(* PLC project Base_Elements, Beckhoff Automation GmbH TwinCAT PLC Control 3.5.6.0 *)
(* stored: creationDateTime 2015-09-07T10:33:48.4706416, modificationDateTime 2015-09-07T10:33:48.472642 *)

TYPE E_ADS_AccessType : (READ := 0, WRITE := 1);
END_TYPE

TYPE T_ADS_ConnectionData : STRUCT
  udiConID : UDINT;  (* Connection ID. Automatically assigned by calling method for adding new connection *)
  udiHandle : UDINT;  (* Handle ID for data exchange. Determined automatically during state PONbusy. *)
  strRoute : STRING;  (* Route of the PRG or FUB instance on server side. Example: 'SlowPRG_1.fbData.SIf.cur.st_ADSData' *)
  uinTargetPort : UINT;  (* ADS target port *)
  strNetID : STRING(30);  (* NetID *)
  eAccessType : E_ADS_AccessType;  (* Access type *)
  udiDataLen : UDINT;  (* Length of the data structure *)
  pData : PVOID;  (* Pointer to data structure. Note: Defined structure must be the same on client and server side. *)
END_STRUCT;
END_TYPE

TYPE T_Ctrl_SIf_ACL : STRUCT
  Par : T_Ctrl_SIf_ACL_Par;  (* parameter *)
  Cur : T_Ctrl_SIf_ACL_Cur;  (* current values *)
  Alm : ARRAY[1..7] OF T_Ctrl_Alm;  (* alarm number used in this controller *)
END_STRUCT;
END_TYPE

TYPE T_Ctrl_SIf_ACL_Cur : STRUCT
  uinNumOfAdsConnections : UINT;  (* Shows the number of ADS (server) connections *)
END_STRUCT;
END_TYPE

TYPE T_Ctrl_SIf_ACL_Par : STRUCT
  udiTOPowerOn_ms : UDINT;  (* [ms] Timeout power on. Timeout for initialize all ADS connections. *)
  udiTOAddRoute_ms : UDINT;  (* [ms] Timeout add route *)
  udiTOReadData_ms : UDINT;  (* [ms] Timeout read data *)
  udiTOWriteData_ms : UDINT;  (* [ms] Timeout write data *)
  udiTORWData_ms : UDINT;  (* [ms] Timeout read/write data *)
  udiPollingInterval_ms : UDINT;  (* [ms] Polling interval for read/write of all ADS connections in list *)
END_STRUCT;
END_TYPE

TYPE E_BCD_Type : (None := 0, SICK, KEYENCE);
END_TYPE

TYPE T_BCD : STRUCT
  strState : STRING;
  strCmd : STRING;
  intCmd : INT;
  stStatus : T_BCD_Status;
  stErr : T_BCD_Error;
  stCfg : T_BCD_Cfg;
  stPar : T_BCD_Par;
  stData : T_BCD_Data;
END_STRUCT;
END_TYPE

TYPE T_BCD_Cfg : STRUCT
  bolSimulation : BOOL;
  strSensorIPAdr : STRING(15) := '';
  udiSensorPort : UDINT := 0;
  iSensorType : E_BCD_Type;
  bolResponseIncludingDiagnostics : BOOL;  (* Barcode is also sending diagnostics data *)
END_STRUCT;
END_TYPE

TYPE T_BCD_Data : STRUCT
  bolCodeReaded : BOOL;
  uliBarCode : ULINT;
  strBarCode : STRING;
  stDevInfo : T_BCD_DeviceInfo;
  stServInfo : T_BCD_ServiceInfo;
  stOpData : T_BCD_OperatingData;
END_STRUCT;
END_TYPE

TYPE T_BCD_DeviceInfo : STRUCT
  strComTestResult : STRING(40);
  strManufacturer : STRING(25);
  strDeviceType : STRING(25);
  strOrderNumber : STRING(20);
  strSWVersion : STRING(10);
  strFWVersion : STRING(10);  (* shows the firmware version of the device *)
  strSerialNumber : STRING(20);
END_STRUCT;
END_TYPE

TYPE T_BCD_Error : STRUCT
  bolErrAck : BOOL;  (* Reset failure *)
  bolErrorActive : BOOL;  (* atleast one failure active *)
  bolSocketError : BOOL;  (* error in TCP socket *)
  bolSensorError : BOOL;  (* error in sensor (SICK) *)
  udiErrorID : UDINT;  (* error ID *)
END_STRUCT;
END_TYPE

TYPE T_BCD_OperatingData : STRUCT
  strPowerOnCounter : STRING(25);
  strOpHours : STRING(25);
  strPowerOnHours : STRING(20);
END_STRUCT;
END_TYPE

TYPE T_BCD_Par : STRUCT
  tTOConnection : TIME;
  tTOSend : TIME;
  tTOReceive : TIME;
END_STRUCT;
END_TYPE

TYPE T_BCD_ServiceInfo : STRUCT
  strLastUsername : STRING(25);
  strLastParChangeDate : STRING(10);
  strLastParChangeTime : STRING(5);
END_STRUCT;
END_TYPE

TYPE T_BCD_StateMachine : STRUCT
  intState : INT;  (* actual state *)
  intStateLastCycle : INT;  (* state of last cycle *)
  intStateHistory : INT;  (* save history backup p.e. in ERROR state *)
  intStateNext : INT;  (* set state for next cycle *)
  udiTimeInState_ms : UDINT;  (* Time in this State *)
END_STRUCT;
END_TYPE

TYPE T_BCD_Status : STRUCT
  bolSocketConnected : BOOL;  (* Socket connected *)
  bolComChecked : BOOL;
END_STRUCT;
END_TYPE

TYPE T_BCD_TxStructure : STRUCT
  intMessageSize : UINT;  (* Actual message size *)
  aTxData : ARRAY[0..300] OF BYTE;  (* Tx data buffer *)
END_STRUCT;
END_TYPE

TYPE E_ALM_PRS : (Dummy := 1, MAX_E_ALM_PRS) UINT;
END_TYPE

TYPE T_Ctrl_SIf_PRS : STRUCT
  Cfg : T_Ctrl_SIf_PRS_Cfg;  (* configuration *)
  Par : T_Ctrl_SIf_PRS_Par;  (* parameter *)
  Cur : T_Ctrl_SIf_PRS_Cur;  (* current values *)
  In : T_Ctrl_SIf_PRS_In;  (* io input *)
  Out : T_Ctrl_SIf_PRS_Out;  (* io output *)
  Alm : ARRAY[1..E_ALM_PRS.MAX_E_ALM_PRS] OF T_Ctrl_Alm;  (* alarm number used in this controller *)
  Ilk : T_Ctrl_SIf_PRS_Ilk;  (* interlock of output/movements *)
END_STRUCT;
END_TYPE

TYPE T_Ctrl_SIf_PRS_Cfg : STRUCT

END_STRUCT;
END_TYPE

TYPE T_Ctrl_SIf_PRS_Cur : STRUCT

END_STRUCT;
END_TYPE

TYPE T_Ctrl_SIf_PRS_Ilk : STRUCT

END_STRUCT;
END_TYPE

TYPE T_Ctrl_SIf_PRS_In : STRUCT
  bolPresent : BASE_PLC.T_Ctrl_IoBool;  (* Input Sensor is present *)
END_STRUCT;
END_TYPE

TYPE T_Ctrl_SIf_PRS_Out : STRUCT

END_STRUCT;
END_TYPE

TYPE T_Ctrl_SIf_PRS_Par : STRUCT
  udiDebouncePresentTime_ms : UDINT;  (* [ms] Debounce time until it shows as present *)
  udiDebounceAbsentTime_ms : UDINT;  (* [ms] Debounce time until it shows as absent *)
  bolSimHangerAvailable : BOOL;  (* True = simulated hanger available *)
END_STRUCT;
END_TYPE

TYPE E_Typ_Baudrate : (baud_2400 := 4, baud_4800 := 5, baud_9600 := 6, baud_19200 := 7, baud_38400 := 8, baud_57600 := 9, baud_115200 := 10);
END_TYPE

(* values of E_Typ_Ftim: RF300: Setting for air interface *)

TYPE E_Typ_Ftim : (RF300 := 0, ISO_generall := 1, ISO_infineon := 3, ISO_Fujitsu := 4, ISO_NXP := 5, ISO_TI := 6, ISO_ST := 7, Max_E_Typ_Ftim);
END_TYPE

TYPE T_RFD : STRUCT
  strState : STRING;
  strCmd : STRING;
  intCmd : INT;
  intServiceCmd : INT;
  stStatus : T_RFD_Status;
  stCfg : T_RFD_Cfg;
  stCur : T_RFD_Cur;
  stErr : T_RFD_Error;
END_STRUCT;
END_TYPE

TYPE T_RFD_Cfg : STRUCT
  bolSimulation : BOOL;
  eTyp : E_Typ_RFW;
  usiResetParameter : USINT := 2#101010;  (* Reset parameter value *)
  usiFtimSetting : E_Typ_Ftim;  (* Setting of the Air interface *)
  usiResetOption1 : USINT := 2#10;  (* Reset option1 value *)
  uinBaudrate : USINT;  (* Set Baudrate *)
  uinComSettings : USINT;  (* Set Communikationsettings *)
  stNetId : TC2_SYSTEM.T_AmsNetID;  (* Net ID oft EtherCat Master *)
  uinSlaveAddr : UINT;  (* Port Number of EtherCat Slave Comunication Module *)
  uinCoeIndexComSettings : WORD := 16#8000;  (* CoE Object Index for Communication Settings *)
  usiCoeSubindexComBaudrate : BYTE := 16#11;  (* CoE Object SubIndex for Baudrate *)
  usiCoeSubindexComDataframe : BYTE := 16#15;  (* CoE Object SubIndex for Dataframe *)
  udiRetry : UDINT := 10;  (* Retry Job to RFID Reader *)
  usiMemory : USINT := 0;  (* /////////////////////////////////////////////// Reset Memory 00=RAM, 01=remanent *)
  usiScanMode : USINT := 1;  (* Scan Mode 00= Continous Read; 01=Single Read *)
  uinLockTime_ms : UINT := 5000;  (* Lock Time in ms *)
END_STRUCT;
END_TYPE

TYPE T_RFD_Cur : STRUCT
  pData : POINTER TO ARRAY[0..255] OF BYTE;  (* Pointer to Received Data Array *)
  uinAdressData : UINT;  (* Startadress to Read/Write at the data Array Element *)
  uinAdressTag : UINT;  (* Startadress to Read/Write at the Tag *)
  usiCount : USINT;  (* Number of bytes to Read/Write *)
END_STRUCT;
END_TYPE

TYPE T_RFD_Error : STRUCT
  bolErrAck : BOOL;  (* Reset failure *)
  bolErrorActive : BOOL;  (* atleast one failure active *)
  bolComError : BOOL;  (* error at communication card *)
  bolProtcolError : BOOL;
  bolRFIDError : BOOL;  (* Error with RF ID Tag *)
  bolSDOError : BOOL;  (* Error at setting of the communication Card (SDO Write) *)
  udiErrorID : UDINT;  (* information to Communication Card error *)
END_STRUCT;
END_TYPE

TYPE T_RFD_MDS_Diagnose : STRUCT
  usiLFD : USINT;  (* Power flux density: as smaller the value, as higher the field intensity *)
  usiFZP : USINT;  (* Errorcounter inactive mode *)
  usiFZA : USINT;  (* Errorcounter active: CRC or signature errors *)
  usiANWZ : USINT;  (* Presence time of tag, resolution in 9.7ms *)
END_STRUCT;
END_TYPE

TYPE T_RFD_MDS_State : STRUCT
  bytMDSType : BYTE;  (* MDS Type 1=no FRAM; 2=8k FRAM; 3=32k FRAM; 4=64k FRAM; 5=128k FRAM; 6=256k FRAM *)
  bytLockState : BYTE;  (* Lock bit registers (lock state) *)
  bytVersion : BYTE;  (* MDS Version *)
  worMemSize : WORD;  (* Memory Size *)
  bytBlockSize : BYTE;  (* Blocksize in Byte *)
  bytBlockNo : BYTE;  (* Value of memory Blocks *)
END_STRUCT;
END_TYPE

TYPE T_RFD_SLG_Diagnose : STRUCT
  usiS_Info : USINT;  (* Mode SLG Diagnose *)
  usiFZP : USINT;  (* Errorcounter inactive mode *)
  usiABZ : USINT;  (* Counter abort *)
  usiCFZ : USINT;  (* Errorcounter code errors *)
  usiSFZ : USINT;  (* Errorcounter signature errors *)
  usiCRCFZ : USINT;  (* Errorcounter CRC *)
  usiBSTAT : USINT;  (* Actual command state *)
  usiASMFZ : USINT;  (* Counter interface errors to host (Parity, BCC, Frame) *)
END_STRUCT;
END_TYPE

TYPE T_RFD_SLG_State : STRUCT
  bytHWType : BYTE;  (* HW Type of SLG 0=RF310R RF340R RF350R (-xAA10); 1=RF380R (-3AA10); 2=RF310R(-1AB10); 3=RF380R (-3AB10); 4=RF340R RF350R (-2AB10,-4AB10) *)
  worHWVersion : WORD;  (* HW Version *)
  worURLVersion : WORD;  (* Loading Version *)
  bytFWType : BYTE;  (* FW Type *)
  worFWVersion : WORD;  (* FW Version *)
  bytDriverType : BYTE;  (* Driver Type 1=3964R *)
  worDriverVersion : WORD;  (* Driver Version *)
  bytComm : BYTE;  (* Communication port 1=RS422, 2=RS232 *)
  bytBaud : BYTE;  (* Communication Baud rate 1=19.2kBaud; 3=57.6kBaud; 5=115.2kBaud *)
  bytPower : BYTE;  (* sending power (only RF380R) 0=standard; 2=0.5W; 3=0.75W; 4=1W; 5=1.25W (default); 6=1.5W; 7=1.75W; 8=2W *)
  bytMtag : BYTE;  (* Number of maximal tags in the field *)
  bytFtim : BYTE;  (* air interface 0=RF300; 1=ISO generall; 3=ISO infineon Chip; 4=ISO Fujitsu; 5=ISO NXP; 6=ISO TI; 7=ISO ST *)
  bytAntenna : BYTE;  (* State antenna 1=ON; 2=OFF *)
  bytPresence : BYTE;  (* Tag presence 0=No presence; 1=prexence *)
END_STRUCT;
END_TYPE

TYPE T_RFD_StateMachine : STRUCT
  intState : INT;  (* actual state *)
  intStateLastCycle : INT;  (* state of last cycle *)
  intStateHistory : INT;  (* save history backup p.e. in ERROR state *)
  intStateNext : INT;  (* set state for next cycle *)
  udiTimeInState_ms : UDINT;  (* Time in this State *)
END_STRUCT;
END_TYPE

TYPE T_RFD_Status : STRUCT
  bolStartupOk : BOOL;  (* 1 = Antenna is initialized *)
  bolInitOk : BOOL;  (* 1 = Antenna is initialized *)
  bolOn : BOOL;  (* 1 = Antenna is on *)
  bolPresent : BOOL;  (* 1 = tag is present *)
  bolL_UEB : BOOL;  (* 1 = Communication to SLG is OK *)
  stSLG_State : T_RFD_SLG_State;  (* SLG State only actual on demand *)
  stSLG_Diag : T_RFD_SLG_Diagnose;  (* SLG Diagnose only actual on demand *)
  stMDS_State : T_RFD_MDS_State;  (* SLG State only actual on demand *)
  stMDS_Diag : T_RFD_MDS_Diagnose;  (* SLG Diagnose only actual on demand *)
  abyteUID : ARRAY[0..7] OF BYTE;  (* Tag ID *)
END_STRUCT;
END_TYPE

TYPE T_StateWord : STRUCT
  bolTransmitAccepted : BOOL;  (* Acknowledge the datachange of this Command bit *)
  bolReceiveRequest : BOOL;  (* New Datat at the input *)
  bolInputAccepted : BOOL;  (* 0=Ready for Data exchange; 1=initialisation of the clam *)
  bolBufferFull : BOOL;  (* Input Buffer is full, all new arriveing data lost *)
  bolParityErr : BOOL;  (* Parity Error occured *)
  bolFramingErr : BOOL;  (* Framing Error occured *)
  bolOverrunErr : BOOL;  (* Overrun Error occured *)
  usiInLenght : USINT;  (* Amounth of the reached Input Bytes *)
END_STRUCT;
END_TYPE

TYPE E_LIGHTSTATE : (Off, BlinkSlow, BlinkFast, On);
END_TYPE

TYPE E_StackLightColor : (Red, Yellow, Green, Blue, Max_SackLightColor);
END_TYPE

TYPE T_LighInformation : STRUCT
  eState : E_LIGHTSTATE;
  udiTime_ms : UDINT;
  bolOutput : REFERENCE TO REFERENCE TO BOOL;
END_STRUCT;
END_TYPE

TYPE T_BCC_Data : STRUCT
  uliBarCode : ULINT;
  strBarCode : STRING;
END_STRUCT;
END_TYPE

TYPE T_Ctrl_SIf_BCC : STRUCT
  Cfg : T_Ctrl_SIf_BCC_Cfg;  (* configuration *)
  Par : T_Ctrl_SIf_BCC_Par;  (* parameter *)
  Cur : T_Ctrl_SIf_BCC_Cur;  (* current values *)
  In : T_Ctrl_SIf_BCC_In;  (* io input *)
  Out : T_Ctrl_SIf_BCC_Out;  (* io output *)
  Alm : ARRAY[1..7] OF T_Ctrl_Alm;  (* alarm number used in this controller *)
END_STRUCT;
END_TYPE

TYPE T_Ctrl_SIf_BCC_Cfg : STRUCT
  strSensorIPAdr : STRING(15) := '';  (* IP Adress of the sensor (PLC = Client, Sensor = Server) *)
  udiSensorPort : UDINT := 0;  (* Port number of the sensor *)
  iSensorType : E_BCD_Type;
END_STRUCT;
END_TYPE

TYPE T_Ctrl_SIf_BCC_Cur : STRUCT
  bolConnected : BOOL;  (* Sensor connected *)
  bolComChecked : BOOL;  (* Communication checked during PON *)
  bolNewCodeReaded : BOOL;  (* 1 = new bar code readed *)
  bolNoRead : BOOL;  (* 1 = no code readed, answer *No Read* *)
  stData : T_BCC_Data;  (* Sensor data *)
END_STRUCT;
END_TYPE

TYPE T_Ctrl_SIf_BCC_In : STRUCT
  bolSensorTrigScan : BASE_PLC.T_Ctrl_IoBool;  (* Sensor input for triggering a new barcode scan *)
END_STRUCT;
END_TYPE

TYPE T_Ctrl_SIf_BCC_Out : STRUCT

END_STRUCT;
END_TYPE

TYPE T_Ctrl_SIf_BCC_Par : STRUCT
  udiTOPowerOn_ms : UDINT;  (* [ms] Timeout power on *)
  udiTORead_ms : UDINT;  (* [ms] Timeout read *)
  udiExecuteScanDelayTime_ms : UDINT;  (* [ms] Barcode scan delay time - Delay before a barcode scan will be triggered after a new product has been detected by trigger sensor input *)
END_STRUCT;
END_TYPE

{attribute 'qualified_only'}
TYPE E_ALM_CYL : (SensorRetractAlwaysOn := 1, SensorExtendNotReached := 2, SensorExtendAlwaysOn := 3, SensorRetractNotReached := 4, InterlockExtend := 5, InterlockRetract := 6, MAX_E_ALM) UINT;
END_TYPE

(* values of E_Typ_CYL: Valve2_Sensor2: bistabile and two feedback sensors; Valve2_SensorExtended: bistabile and extended feedback sensors; Valve2_SensorRetracted: bistabile and retracted feedback sensors; Valve2_Sensor0: bistabile and no feedback sensors; Valve1_Sensor2: monostabile and 2 feedback sensors; Valve1_SensorExtended: monostabile and extended feedback sensors; Valve1_SensorRetracted: monostabile and retracted feedback sensor; Valve1_Sensor0: monostabile and no feedback sensors *)

TYPE E_Typ_CYL : (Valve2_Sensor2 := 0, Valve2_SensorExtended, Valve2_SensorRetracted, Valve2_Sensor0, Valve1_Sensor2, Valve1_SensorExtended, Valve1_SensorRetracted, Valve1_Sensor0, Max_E_Typ_CYL);
END_TYPE

TYPE T_Ctrl_SIf_CYL : STRUCT
  Cfg : T_Ctrl_SIf_CYL_Cfg;  (* configuration *)
  Par : T_Ctrl_SIf_CYL_Par;  (* parameter *)
  Cur : T_Ctrl_SIf_CYL_Cur;  (* current values *)
  In : T_Ctrl_SIf_CYL_In;  (* io input *)
  Out : T_Ctrl_SIf_CYL_Out;  (* io output *)
  Alm : ARRAY[1..(E_ALM_CYL.MAX_E_ALM - 1)] OF T_Ctrl_Alm;  (* alarm number used in this controller *)
  Ilk : T_Ctrl_SIf_CYL_Ilk;  (* interlock of output/movements *)
END_STRUCT;
END_TYPE

TYPE T_Ctrl_SIf_CYL_Cfg : STRUCT
  eTyp : E_Typ_CYL;
END_STRUCT;
END_TYPE

TYPE T_Ctrl_SIf_CYL_Cur : STRUCT
  udiMoveTimeRetract : UDINT;  (* [ms] time last movement to retract *)
  udiMoveTimeExtend : UDINT;  (* [ms] time last movement to extend *)
END_STRUCT;
END_TYPE

TYPE T_Ctrl_SIf_CYL_Ilk : STRUCT
  bolRetract : BOOL;  (* interlock retraction of cylinder *)
  bolExtend : BOOL;  (* interlock extend of cylinder *)
END_STRUCT;
END_TYPE

TYPE T_Ctrl_SIf_CYL_In : STRUCT
  bolExtended : T_Ctrl_IoBool;  (* sensor feedback position extended reached *)
  bolRetracted : T_Ctrl_IoBool;  (* sensor feedback position retracted reached *)
END_STRUCT;
END_TYPE

TYPE T_Ctrl_SIf_CYL_Out : STRUCT
  bolRetract : T_Ctrl_IoBool;  (* switch valve retract *)
  bolExtend : T_Ctrl_IoBool;  (* switch valve extend *)
END_STRUCT;
END_TYPE

TYPE T_Ctrl_SIf_CYL_Par : STRUCT
  udiExtendTime_ms : UDINT;  (* [ms] until failure to long time for extend *)
  udiRetractTime_ms : UDINT;  (* [ms] until failure to long time for retract *)
  udiSimExtendTime_ms : UDINT;  (* [ms] simulation time for extend or /2 of timeout time? *)
  udiSimRetractTime_ms : UDINT;  (* [ms] simulation time for retract or /2 of timeout time? *)
END_STRUCT;
END_TYPE

TYPE E_Typ_DRV : (None := 0, TLP, TLK, TLKV, TLPsort, TLS, TLC, Max_E_Typ_JUN);
END_TYPE

TYPE T_Ctrl_SIf_DRV : STRUCT
  Cfg : T_Ctrl_SIf_DRV_Cfg;  (* configuration *)
  Par : T_Ctrl_SIf_DRV_Par;  (* parameter *)
  Cur : T_Ctrl_SIf_DRV_Cur;  (* current values *)
  In : T_Ctrl_SIf_DRV_In;  (* io input *)
  Out : T_Ctrl_SIf_DRV_Out;  (* io output *)
  Alm : ARRAY[1..5] OF T_Ctrl_Alm;  (* alarm number used in this controller *)
END_STRUCT;
END_TYPE

TYPE T_Ctrl_SIf_DRV_Cfg : STRUCT
  eTyp : E_Typ_DRV;  (* Type of drive *)
  dinDistPerPulse_um : DINT;  (* Distance per pulse *)
  bolSpeedVariable : BOOL;  (* Has Variable Speed *)
  bolPulseExist : BOOL;  (* Has Pulse signal for position and speed calculation *)
  usiCountBlockedSupervis : USINT;  (* Number of blocked supervision inputs *)
  dinPinDistance_um : DINT;  (* [um] PinDistance *)
  bolEnableMaintenaceSwitch : BOOL;  (* Enable Maintenace Switch *)
END_STRUCT;
END_TYPE

TYPE T_Ctrl_SIf_DRV_Cur : STRUCT
  dinPulseCounter : DINT;
  dinPos_um : DINT;
  dinSpeed_um_s : DINT;
END_STRUCT;
END_TYPE

TYPE T_Ctrl_SIf_DRV_In : STRUCT
  bolOverload : T_Ctrl_IoBool;
  bolPulse : T_Ctrl_IoBool;
  a_bolBlockedSupvervis : ARRAY[1..cMAX_BLOCKED_SUP] OF BASE_PLC.T_Ctrl_IoBool;
  bolMaintenanceSwitch : T_Ctrl_IoBool;  (* DI of Maintenance Switch *)
END_STRUCT;
END_TYPE

TYPE T_Ctrl_SIf_DRV_Out : STRUCT
  bolSpeed_1 : T_Ctrl_IoBool;  (* bolSpeed_1 = slow bolSpeed_2 = fast bolSpeed_1 & bolSpeed_2 = middle speed *)
  bolSpeed_2 : T_Ctrl_IoBool;
END_STRUCT;
END_TYPE

TYPE T_Ctrl_SIf_DRV_Par : STRUCT
  udi_pulseTimeout_ms : UDINT;  (* [ms] Timeout supervision of pulse in RUN *)
  udi_pulseSim_ms : UDINT;  (* [ms] Simulation of pulse in RUN: 0.676mm/ms / 38.4mm/puls => 56.8ms/puls *)
  usi_speedLevel : USINT;  (* 0=slow, 1=middle, 2=fast *)
  int_MaxBrokenPins : INT;  (* Maximum Broken Pins *)
END_STRUCT;
END_TYPE

(* values of E_ALM_ECD: ADS_ComError: ADS Communication Error to EtherCAT Master => Info = ADS_Errorcode; TimeOutFunction: A Function is not finished after the defined Timeout; NotAllSlaveConnected: Configured and reached Slaves are not the same => Info Byte 0+1 = Slave Addres from last error Info Byte 2+3 = Numbers of error Slaves; ToManySlaves: More slaves at the master as the structure could handle => Info Byte 0+1 = Slave Addres from last error Info Byte 2+3 = Numbers of error Slaves; MasterStateError: Master not in the correct state => Info = Masterstate; SlaveStateError: Minimum one Slave not in the correct state => Byte 0+1 = Slave Addres from last error, Info Byte 2 + 3 = State of last error Slave; SlaveCRCError: Minimum one Slave has to many CRC Erros => Byte 0+1 = Slave Addres from last error, Info Byte 2 +3 = Number of CRC Errors from last Slave with error; SlaveLinkError: Minimum one Slave has a LinkState Erros => Byte 0+1 = Slave Addres from last error Info Byte 2 + 3 = Link State of last error Slave; NoSlaveFound: No slave found in the network; StateChanges: To many abnormal State Changes *)

TYPE E_ALM_ECD : (ADS_ComError := 1, TimeOutFunction := 2, NotAllSlaveConnected := 3, ToManySlaves := 4, MasterStateError := 5, SlaveStateError := 6, SlaveCRCError := 7, SlaveLinkError := 8, NoSlaveFound := 9, StateChanges := 10, MAX_E_ALM) UINT;
END_TYPE

TYPE T_Ctrl_SIf_ECD : STRUCT
  Cfg : T_Ctrl_SIf_ECD_Cfg;  (* configuration *)
  Par : T_Ctrl_SIf_ECD_Par;  (* parameter *)
  Cur : T_Ctrl_SIf_ECD_Cur;  (* current values *)
  Alm : ARRAY[1..(E_ALM_ECD.MAX_E_ALM - 1)] OF T_Ctrl_Alm;  (* alarm number used in this controller *)
END_STRUCT;
END_TYPE

TYPE T_Ctrl_SIf_ECD_Cfg : STRUCT
  strNetID : STRING(30);  (* NetID *)
  bolRunAlways : BOOL;  (* Run allways the scanning without set into run *)
END_STRUCT;
END_TYPE

TYPE T_Ctrl_SIf_ECD_Cur : STRUCT
  uinNumOfSlaves : UINT;  (* Shows the number of EtherCAT Slaves *)
  stSlaveData : ARRAY[0..ECD_Const.cuinMaxSlaves] OF T_ECD_SlaveData;  (* Information of every slave *)
  worMasterState : WORD;  (* State Of Master *)
  udiCRCSumm : UDINT;  (* All CRC Errors *)
  uinNumOfSlaveErrors : UINT;  (* Counter of Slave Errors State *)
END_STRUCT;
END_TYPE

TYPE T_Ctrl_SIf_ECD_Par : STRUCT
  udiTOPowerOn_ms : UDINT;  (* [ms] Timeout power on. Timeout for initialize all ADS connections. *)
  udiTOCheckAll_ms : UDINT;  (* [ms] Timeout function over all slaves *)
  udiTOCheckOne_ms : UDINT;  (* [ms] Timeout function for one slave *)
  udiPollingInterval_ms : UDINT;  (* [ms] Polling interval for States *)
  udiMaxCRC : UDINT;  (* Maximum CRC Value one slave *)
END_STRUCT;
END_TYPE

TYPE T_ECD_SlaveData : STRUCT
  stConfigData : Tc2_EtherCAT.ST_EcSlaveConfigData;  (* Slave Configuration *)
  uinAddress : UINT;  (* Address of the slave (as UINT, beacuase in stConfigData is only as WORD) *)
  stState : Tc2_EtherCAT.ST_EcSlaveState;  (* State of the slave *)
  stCRCError : Tc2_EtherCAT.ST_EcCrcErrorEx;  (* CRC Error totally *)
END_STRUCT;
END_TYPE

(* values of E_Typ_RFW: RF310R: RF310; RF382R: RF382R *)

TYPE E_Typ_RFW : (RF310R := 0, RF382R := 1, Max_E_Typ_CYL);
END_TYPE

TYPE T_Ctrl_SIf_RFW : STRUCT
  Cfg : T_Ctrl_SIf_RFW_Cfg;  (* configuration *)
  Par : T_Ctrl_SIf_RFW_Par;  (* parameter *)
  Cur : T_Ctrl_SIf_RFW_Cur;  (* current values *)
  In : T_Ctrl_SIf_RFW_In;  (* io input *)
  Out : T_Ctrl_SIf_RFW_Out;  (* io output *)
  DtChnToLine : T_Ctrl_SIf_RFW_DtChnToLine;  (* Data Channel from PLC to Line Controller *)
  Alm : ARRAY[1..6] OF T_Ctrl_Alm;  (* alarm number used in this controller *)
END_STRUCT;
END_TYPE

TYPE T_Ctrl_SIf_RFW_Cfg : STRUCT
  eTyp : E_Typ_RFW;
  bolGetTrayIDAuto : BOOL;  (* Get automatically the Tray ID too *)
  stNetId : TC2_SYSTEM.T_AmsNetID;  (* Net ID oft EtherCat Master *)
  uinSlaveAddr : UINT;  (* Port Number of EtherCat Slave Comunication Module *)
  bolDtChToLine_send : BOOL;  (* Send every New RFID to Line controller *)
END_STRUCT;
END_TYPE

TYPE T_Ctrl_SIf_RFW_Cur : STRUCT
  bolPresent : BOOL;  (* 1 = tag is present *)
  abytData : ARRAY[0..255] OF BYTE;  (* Data to read / write *)
  stData : T_RFW;  (* Data in Structure *)
  dwoJob : DWORD;  (* Job information, what data read or write *)
END_STRUCT;
END_TYPE

TYPE T_Ctrl_SIf_RFW_DtChnToLine : STRUCT
  stNewRfid : T_NewRFID_DtChn;
END_STRUCT;
END_TYPE

TYPE T_Ctrl_SIf_RFW_In : STRUCT

END_STRUCT;
END_TYPE

TYPE T_Ctrl_SIf_RFW_Out : STRUCT

END_STRUCT;
END_TYPE

TYPE T_Ctrl_SIf_RFW_Par : STRUCT
  udiReadTime_ms : UDINT;  (* [ms] until failure to long time for read *)
  udiWriteTime_ms : UDINT;  (* [ms] until failure to long time for write *)
  udiMinCmdTime : UDINT;  (* [ms] minimum wait time between two read command *)
  udiLockTime : UDINT;  (* [ms] locktime prevents sending same ID's to LineControl multiple times *)
END_STRUCT;
END_TYPE

TYPE T_NewRFID_DtChn : STRUCT
  strID : STRING;  (* configurable if Tag or Tray ID *)
  uliTagID : ULINT;
  strTimestamp : STRING(24);
  intDataState : INT;
END_STRUCT;
END_TYPE

TYPE T_RFW : STRUCT
  usiRepetitionID : USINT;  (* Repeteition ID Identifies the try number in the sequence *)
  bolWorkstation2 : BOOL;  (* Workstation 2 workstations in the cell 1 BIT 0: Workstation1, 2: Workstation2 *)
  bolDeleteFileAfterPrint : BOOL;  (* usiProductID : USINT; // The product ID bits 1 to 5 are indeed not used. Mail T.Bosgiraud 11.6.2013 Product type Max number of product types = 32 5 bits, product ID (bits 1 to 5), *)
  bolPrintOk : BOOL;  (* 1 means that the image has been printed without problem. *)
  bolHeightUseMeasure : BOOL;  (* 0: Use the bottom of the tray as basis and add Offset *)
  usiHeightOffset : USINT;  (* Email 1.06.2013 Berk “Use measured height=1”, the actual measurement of the laser plus any offsets programmed into the tray are used to adjust the lifting height 1: Use the printable product surface as basis and add Offset to the measured height *)
  bolHeightOffsetSignMinus : BOOL;  (* “Offset +/-” = 1 means that the printable surface OF the item will go further away FROM the print head. *)
  bolIonizer : BOOL;  (* “Offset +/-” = 0 (default value) means that the printable surface of the item will come closer to the print head *)
  usiPlasmaLevel : USINT;  (* Pre-treatment Plasma 0: Plasma off, 1: Level 1 ..3:Level3 *)
  bolPrintPass : BOOL;  (* Print numbers 1 means that the image needs to be printed twice on the products *)
  bolNozzleCheck : BOOL;  (* 1 means that the nozzle check pattern has to be printed onto the products. *)
  bolAligneCheck : BOOL;  (* 1 means that the alignment check pattern has to be printed onto the products. *)
  usiUVPinningLevel : USINT;  (* UV-pinning intensity 0: Level1 ... 15: Level16 *)
  usiUVLampLevel : USINT;  (* UV-lamp intensity 0: Level1 ... 15: Level16 *)
  strFileName : STRING;  (* p.e.: 268205625-3.pdf -> The file name sent by VIPER to the printer and to the conveyor is made out of 64 bits *)
  bolBrush : BOOL;  (* The RFID divides the rest of the name (268205625-3) as 8 successive bytes arranged as follows: - Byte 7 (RFID byte 0Dhex) to byte 1 (RFID byte 07hex) express the number before the hyphen sign (in this case 268205625) - Byte 0 (RFID byte 06hex) expresses the number after the hyphen sign (in this case 3). *)
  bolBrushClean : BOOL;  (* 1: use second brush means that the brush has TO be used FOR the considered tray *)
  bolBrushFans : BOOL;  (* “Brush Fans”=1 means that the fans have to be used for the considered tray *)
  bolGutterClean : BOOL;  (* “Gutter Clean”=1 means that the tray is running for gutter cleaning purposes. *)
  bolSpecialTray : BOOL;  (* This bit tells whether the tray is a regular production tray or a special tray (nozzle check, alignment...). *)
  strTrayID : STRING;  (* Byte 0-13 ->9999999999999 *)
  strTagID : STRING;  (* Byte 0-13 ->9999999999999 *)
  uliTagID : ULINT;
END_STRUCT;
END_TYPE

{attribute 'qualified_only'}
TYPE E_ALM_SGT : (Dummy := 1, MAX_E_ALM) UINT;
END_TYPE

TYPE T_Ctrl_SIf_SGT : STRUCT
  Cfg : T_Ctrl_SIf_SGT_Cfg;  (* configuration *)
  Par : T_Ctrl_SIf_SGT_Par;  (* parameter *)
  Out : T_Ctrl_SIf_SGT_Out;  (* io output *)
  Alm : ARRAY[1..(E_ALM_SGT.MAX_E_ALM - 1)] OF T_Ctrl_Alm;  (* alarm number used in this controller *)
END_STRUCT;
END_TYPE

TYPE T_Ctrl_SIf_SGT_Cfg : STRUCT
  bolEnableLampTest : BOOL;  (* Enable lamp test in PONBusy state *)
END_STRUCT;
END_TYPE

TYPE T_Ctrl_SIf_SGT_Out : STRUCT
  bolGreen : T_Ctrl_IoBool;  (* green lamp *)
  bolYellow : T_Ctrl_IoBool;  (* yellow lamp *)
  bolRed : T_Ctrl_IoBool;  (* red lamp *)
  bolBeep : T_Ctrl_IoBool;  (* acoustic signal *)
END_STRUCT;
END_TYPE

TYPE T_Ctrl_SIf_SGT_Par : STRUCT
  udiBlinkTime_ms : UDINT;  (* [ms] Blink interval time *)
  udiBeepOnTime_ms : UDINT;  (* [ms] Beep on time *)
  udiBeepOffTime_ms : UDINT;  (* [ms] Beep off time *)
  udiLampTestTime_ms : UDINT;  (* [ms] Lamp test time, used in PONBusy *)
END_STRUCT;
END_TYPE

TYPE E_ALM_UMC : (MotorOnTimeout := 1, MotorError := 2, MotorWarning := 3, MotorOverCurrent := 4, MotorNotReady := 5, DirectionParameterOverflow := 6, SpeedOverLimit := 7, MotorStatusInformation := 8, MAX_E_ALM_UMC);
END_TYPE

TYPE E_CFG_UMC : (Standard := 0, LenzeFC := 1, MAY_E_CFG_UMC);
END_TYPE

TYPE E_TURN_DIRECTION : (AUTOMATIC := 0, LEFT := 1, RIGHT := 2, MAX_E_TURN_DIRECTION);
END_TYPE

TYPE E_UMC_MOTOR_STATUS : (FirmwareUpdate := 0, Init := 1, MotorIdent := 2, ReadyToSwitchON := 3, SwitchedON := 4, OperationEnabled := 5, Warning := 6, Trouble := 7, Fault := 8, TroubleQSP := 9, SafeTorqueOff := 10, SystemFail := 11, MAX_E_UMC_MOTOR_STATUS);
END_TYPE

TYPE T_Ctrl_SIf_UMC : STRUCT
  Cfg : T_Ctrl_SIf_UMC_Cfg;  (* configuration *)
  Par : T_Ctrl_SIf_UMC_Par;  (* parameter *)
  Cur : T_Ctrl_SIf_UMC_Cur;  (* current values *)
  In : T_Ctrl_SIf_UMC_In;  (* io input *)
  Out : T_Ctrl_SIf_UMC_Out;  (* io output *)
  Alm : ARRAY[1..MAX_E_ALM_UMC] OF T_Ctrl_Alm;  (* alarm number used in this controller *)
  Ilk : T_Ctrl_SIf_UMC_Ilk;  (* interlock of output/movements *)
END_STRUCT;
END_TYPE

TYPE T_Ctrl_SIf_UMC_Cfg : STRUCT
  MotorType : E_CFG_UMC;  (* Motor Type *)
  uinLC11 : UINT;  (* [RPM] L0011 Setting of the Lenze motor. This value is 100% of the output control setting. *)
  uinLC11_100 : UINT;  (* Value that is equal to 100% of LC11 *)
  uinMaxSpeed : UINT;  (* Maximum allowed speed in [%] of LC11 *)
END_STRUCT;
END_TYPE

TYPE T_Ctrl_SIf_UMC_Cur : STRUCT
  eDirection : E_TURN_DIRECTION;  (* Actual Turning Direction *)
  uinSpeedOuput : UINT;  (* Actual speed as output 16384 = 100% of L-C11 (1500RPM) *)
  uinSpeed_rpm : UINT;  (* Actual speed as output in [rpm] *)
  uinSpeedLimit : UINT;  (* Motor Limit as Output value *)
  uinMotorResetCnt : UINT;  (* Motor reset retries *)
END_STRUCT;
END_TYPE

TYPE T_Ctrl_SIf_UMC_Ilk : STRUCT

END_STRUCT;
END_TYPE

TYPE T_Ctrl_SIf_UMC_In : STRUCT
  uinStatus : Base_PLC.T_Ctrl_IoUint;  (* Status Word of Lenze *)
  intMotorActualSpeed : Base_PLC.T_Ctrl_IoInt;  (* Motor actual speed *)
  uinMotorSetSpeed : Base_PLC.T_Ctrl_IoUint;  (* Motor actual speed setpoint *)
  bol400V_Ok : Base_PLC.T_Ctrl_IoBool;  (* Motor 400V available information *)
END_STRUCT;
END_TYPE

TYPE T_Ctrl_SIf_UMC_Out : STRUCT
  uinControl : BASE_PLC.T_Ctrl_IoUint;  (* Control word for Lenze FU *)
  uinSpeedSetpoint : BASE_PLC.T_Ctrl_IoUint;  (* Speed Setpoint; 16384 (214) ≡ 100% (bez. auf L-C11) *)
END_STRUCT;
END_TYPE

TYPE T_Ctrl_SIf_UMC_Par : STRUCT
  eRotationDirection : E_TURN_DIRECTION;  (* Rotation direction E_CFG_UMC *)
  udiStartupOnTime_ms : UDINT;  (* [ms] time to initialize and reset the errors on the motor *)
  udiMotorOnTime_ms : UDINT;  (* [ms] time the motor has time to go from OFF to ON *)
  uinSpeed_rpm : UINT;  (* [rpm] Speed control selection *)
  udiSimMotorOnTime_ms : UDINT;  (* [ms] time to wait until the motor reaches the set speed. *)
  udiMoveStartLatency : UDINT;  (* [ms] Delay until the drive startsup *)
  udiMoveStopLatency : UDINT;  (* [ms] Delay until the drive stops *)
  uinMotorResetCnt : UINT;  (* Motor reset retries *)
  uinMotorResetPulseTime_ms : UINT;  (* [ms] Motor Reset Pulse Time *)
END_STRUCT;
END_TYPE

TYPE T_UMC_Lenze_Control : STRUCT
  SwitchOn : BIT;
  DisableVoltage : BIT;
  SetQuickStop : BIT;
  EnableOperation : BIT;
  ModeSpecific_1 : BIT;
  ModeSpecific_2 : BIT;
  ModeSpecific_3 : BIT;
  ResetFault : BIT;
  SetHalt : BIT;
  Reserved_1 : BIT;
  Reserved_2 : BIT;
  SetDCBreak : BIT;
  JogSpeed1 : BIT;
  JogSpeed2 : BIT;
  SetFail : BIT;
  SetSpeedCcw : BIT;
END_STRUCT;
END_TYPE

TYPE T_UMC_Lenze_Status : STRUCT
  FreeStatusBit0 : BIT;
  PowerDisabled_IMP : BIT;
  ImaxActive : BIT;
  SpeedSetReached : BIT;
  SpeedActEqualSet : BIT;
  NActualCompare : BIT;
  ActSpeedIsZero : BIT;
  ControllerInhibit : BIT;
  Status_1 : BIT;
  Status_2 : BIT;
  Status_3 : BIT;
  Status_4 : BIT;
  Warning : BIT;
  Trouble : BIT;
  SpeedCcw : BIT;
  DriveReady : BIT;
END_STRUCT;
END_TYPE

{attribute 'qualified_only'}
TYPE E_ALM_VLV : (SensorOpenAlwaysOn := 1, SensorCloseNotReached := 2, SensorCloseAlwaysOn := 3, SensorOpenNotReached := 4, InterlockOpen := 5, InterlockClose := 6, MAX_E_ALM) UINT;
END_TYPE

(* values of E_Typ_VLV: Valve2_Sensor2: bistabile and two feedback sensors; Valve2_SensorOpened: bistabile and open feedback sensor; Valve2_SensorClosed: bistabile and close feedback sensor; Valve2_Sensor0: bistabile and no feedback sensors; Valve1_Sensor2: monostabile and 2 feedback sensors; Valve1_SensorOpened: monostabile and open feedback sensor; Valve1_SensorClosed: monostabile and close feedback sensor; Valve1_Sensor0: monostabile and no feedback sensors *)

TYPE E_Typ_VLV : (Valve2_Sensor2 := 0, Valve2_SensorOpened, Valve2_SensorClosed, Valve2_Sensor0, Valve1_Sensor2, Valve1_SensorOpened, Valve1_SensorClosed, Valve1_Sensor0, Max_E_Typ_VLV);
END_TYPE

TYPE T_Ctrl_SIf_VLV : STRUCT
  Cfg : T_Ctrl_SIf_VLV_Cfg;  (* configuration *)
  Par : T_Ctrl_SIf_VLV_Par;  (* parameter *)
  Cur : T_Ctrl_SIf_VLV_Cur;  (* current values *)
  In : T_Ctrl_SIf_VLV_In;  (* io input *)
  Out : T_Ctrl_SIf_VLV_Out;  (* io output *)
  Alm : ARRAY[1..(E_ALM_VLV.MAX_E_ALM - 1)] OF T_Ctrl_Alm;  (* alarm number used in this controller *)
  Ilk : T_Ctrl_SIf_VLV_Ilk;  (* interlock of output/movements *)
END_STRUCT;
END_TYPE

TYPE T_Ctrl_SIf_VLV_Cfg : STRUCT
  eTyp : E_Typ_VLV;
END_STRUCT;
END_TYPE

TYPE T_Ctrl_SIf_VLV_Cur : STRUCT
  udiMoveTimeOpen : UDINT;  (* [ms] time last movement to open *)
  udiMoveTimeClose : UDINT;  (* [ms] time last movement to close *)
END_STRUCT;
END_TYPE

TYPE T_Ctrl_SIf_VLV_Ilk : STRUCT
  bolOpen : BOOL;  (* interlock open valve *)
  bolClose : BOOL;  (* interlock close valve *)
END_STRUCT;
END_TYPE

TYPE T_Ctrl_SIf_VLV_In : STRUCT
  bolOpen : T_Ctrl_IoBool;  (* sensor feedback position open reached *)
  bolClose : T_Ctrl_IoBool;  (* sensor feedback position close reached *)
END_STRUCT;
END_TYPE

TYPE T_Ctrl_SIf_VLV_Out : STRUCT
  bolOpen : T_Ctrl_IoBool;  (* switch valve open *)
  bolClose : T_Ctrl_IoBool;  (* switch valve close *)
END_STRUCT;
END_TYPE

TYPE T_Ctrl_SIf_VLV_Par : STRUCT
  udiOpenTime_ms : UDINT;  (* [ms] until failure to long time for open *)
  udiCloseTime_ms : UDINT;  (* [ms] until failure to long time for close *)
  udiSimOpenTime_ms : UDINT;  (* [ms] simulation time for open or /2 of timeout time? *)
  udiSimCloseTime_ms : UDINT;  (* [ms] simulation time for close or /2 of timeout time? *)
END_STRUCT;
END_TYPE

TYPE E_ALM_VPC : (VacuumPumpOnTimeout := 1, VacuumPumpOffTimeout := 2, VacuumFailure := 3, MAX_E_ALM_VPC);
END_TYPE

(* values of E_CFG_VPC: Standard: Only Vacuum Motor with no feedback *)

TYPE E_CFG_VPC : (Standard := 0, VaccumSensor := 1, MotorFeedback := 2, MAY_E_CFG_CYL);
END_TYPE

TYPE T_Ctrl_SIf_VPC : STRUCT
  Cfg : T_Ctrl_SIf_VPC_Cfg;  (* configuration *)
  Par : T_Ctrl_SIf_VPC_Par;  (* parameter *)
  Cur : T_Ctrl_SIf_VPC_Cur;  (* current values *)
  In : T_Ctrl_SIf_VPC_In;  (* io input *)
  Out : T_Ctrl_SIf_VPC_Out;  (* io output *)
  Alm : ARRAY[1..E_ALM_VPC.MAX_E_ALM_VPC] OF T_Ctrl_Alm;  (* alarm number used in this controller *)
  Ilk : T_Ctrl_SIf_VPC_Ilk;  (* interlock of output/movements *)
END_STRUCT;
END_TYPE

TYPE T_Ctrl_SIf_VPC_Cfg : STRUCT
  VacuumPumpFeedback : BOOL;  (* VacuumPump has a feedback *)
  VacuumSensorAvailable : BOOL;  (* Vacuum Sensor available *)
END_STRUCT;
END_TYPE

TYPE T_Ctrl_SIf_VPC_Cur : STRUCT

END_STRUCT;
END_TYPE

TYPE T_Ctrl_SIf_VPC_Ilk : STRUCT

END_STRUCT;
END_TYPE

TYPE T_Ctrl_SIf_VPC_In : STRUCT
  bolVacuumOk : BASE_PLC.T_Ctrl_IoBool;  (* 0 = Vacuum is NOK; 1 = Vacuum is Ok --> Vacuum Pump is probably running *)
  bolPumpOn : BASE_PLC.T_Ctrl_IoBool;  (* Pump has a feedback *)
END_STRUCT;
END_TYPE

TYPE T_Ctrl_SIf_VPC_Out : STRUCT
  bolVacuumPumpOn : BASE_PLC.T_Ctrl_IoBool;  (* 0 = Vacuum Pump Off; 1 = Vacuum Pump On *)
END_STRUCT;
END_TYPE

TYPE T_Ctrl_SIf_VPC_Par : STRUCT
  udiVacuumPumpTime_ms : UDINT;  (* [ms] time the pump has time to go from OFF to ON *)
  udiVacuumStabilizationTime_ms : UDINT;  (* [ms] vacuum stabilization time if no vacuum sensor is available *)
  udiVacuumSensorDebounceTime_ms : UDINT;  (* [ms] time to wait until the vacuum sensor off is acknowledged as off. *)
  udiSimVacuumPumpOnTime_ms : UDINT;  (* [ms] simulation time for Vacuum Pump ON *)
END_STRUCT;
END_TYPE

TYPE E_ALM_MOD : (InvalidPointer := 1, CommunicationError := 2, EmergencyOff := 3, TimeoutStartGroup := 4, TimeoutStopGroup := 5, NextModuleNotReadyWarning := 6, NextModuleNotReadyStop := 7, MAX_E_ALM_MOD) UDINT;
END_TYPE

TYPE E_MOD_STARTUP : (NONE := 0, Start, ReadCsvFile, HostInit, ParameterSync, Ready);
END_TYPE

TYPE T_Ctrl_SIf_MOD : STRUCT
  Cfg : POINTER TO T_Ctrl_SIf_MOD_Cfg;  (* configuration *)
  Par : POINTER TO T_Ctrl_SIf_MOD_Par;  (* parameter *)
  Cur : POINTER TO T_Ctrl_SIf_MOD_Cur;  (* current values *)
  In : POINTER TO T_Ctrl_SIf_MOD_In;  (* io input *)
  Out : POINTER TO T_Ctrl_SIf_MOD_Out;  (* io output *)
  Alm : ARRAY[1..MAX_E_ALM_MOD] OF T_Ctrl_Alm;  (* alarm number used in this controller *)
END_STRUCT;
END_TYPE

TYPE T_Ctrl_SIf_MOD_Cfg : STRUCT
  bolComToLineControlEnabled : BOOL;  (* Enable communication to line control *)
  bolIgnoreReadyInput : BOOL;  (* Ignore Ready Input *)
  bolStackLightHornEnable : BOOL;  (* True = Enable the Stacklight Horn *)
END_STRUCT;
END_TYPE

TYPE T_Ctrl_SIf_MOD_Cur : STRUCT
  dinMaxCapacity : DINT;  (* Max module capacity calculated from all childs which implement interface IBuffer *)
  dinNumOfItems : DINT;  (* Actual number of items calculated from all childs which implement interface IBuffer *)
  bolKeepAliveHost : BOOL;  (* Togglebit set by LineControl to indicate it's still alive. If not, the PLC should stop immediately and wait for LineControl. *)
  bolKeepAlivePlc : BOOL;  (* Togglebit set by PLC to indicate it's still alive. If not, LineControl should stop immediately and try to recover. *)
  a_bBufferIsFull : ARRAY[0..10] OF BOOL;  (* Interface data to LineControl: Indicates that an input port is full. LineControl should not route any more items to this port. *)
  bolStopReleaseItems : ARRAY[0..10] OF BOOL;  (* Interface data from LineControl: Request to stop releasing any item to an output port. The module can still be in RUN state but must not release items to the next module. *)
END_STRUCT;
END_TYPE

TYPE T_Ctrl_SIf_MOD_In : STRUCT
  bolReady : BASE_PLC.T_Ctrl_IoBool;  (* Ready Signal *)
  bolEmoOk : BASE_PLC.T_Ctrl_IoBool;  (* Emo Ok *)
END_STRUCT;
END_TYPE

TYPE T_Ctrl_SIf_MOD_Out : STRUCT
  bolReady : BASE_PLC.T_Ctrl_IoBool;  (* Ready Signal *)
END_STRUCT;
END_TYPE

TYPE T_Ctrl_SIf_MOD_Par : STRUCT
  udiComTimeOutLineCtrl_ms : UDINT;  (* [ms] Communication timeout to line control *)
  aListOfRunGrpWaitTime_ms : ARRAY[0..Base_Const.cMaxNrOfChilds] OF UDINT;  (* [ms] Array with wait time for run groups *)
  aListOfStopGrpWaitTime_ms : ARRAY[0..Base_Const.cMaxNrOfChilds] OF UDINT;  (* [ms] Array with wait time for stop groups *)
  udiTimeoutStopping_ms : UDINT;  (* [ms] timeout for stopping (0= disable timeout monitoring) *)
  udiTimeoutStarting_ms : UDINT;  (* [ms] timeout for starting (0= disable timeout monitoring) *)
END_STRUCT;
END_TYPE

TYPE T_Sequence : STRUCT
  pChild : POINTER TO fb_CtrlBase;
  pCIF : POINTER TO T_Ctrl_CIf;  (* Access to CIF of child *)
  uinGroupRun : UINT;  (* Associated run sequence group *)
  uinGroupStop : UINT;  (* Associated stop sequence group *)
  intCmdSeqRun : INT;  (* Command to be executed for run sequence *)
  intStatusSeqRun : INT;  (* Expected status for run sequence *)
  intStatusSeqRun2 : INT;  (* Alternative status for run sequence *)
  intCmdSeqStop : INT;  (* Command to be executed for run sequence *)
  intStatusSeqStop : INT;  (* Expected status for stop sequence *)
  intStatusSeqStop2 : INT;  (* Alternative status for stop sequence *)
  intCmdSeqStandby : INT;  (* Command to be executed for standby sequence *)
  intStatusSeqStandby : INT;  (* Expected status for standby sequence *)
  intStatusSeqStandby2 : INT;  (* Alternative status for standby sequence *)
  bolChecked : BOOL;  (* Used internal for run and stop sequence to detect if the sequence has been processed *)
END_STRUCT;
END_TYPE

TYPE E_Destination : (StackerA, StackerB, StackerC, Garbage, MAX_E_Destination);
END_TYPE

(* values of E_ItemHealth: Healthy: 0; Ovn_Temperature: 1; Ovn_Time: 2; Ovn_Lost: 3; Hpm_Time: 4; Hpm_Pressure: 5; Hpm_Temperature: 6; Hpm_Lost: 7; Hpm_Unknown: 8; Failed: 9; Lost: 10 - Item is lost somewhere *)

TYPE E_ItemHealth : (Healthy, Ovn_Temperature, Ovn_Time, Ovn_Lost, Hpm_Time, Hpm_Pressure, Hpm_Temperature, Hpm_Lost, Hpm_Unknown, Failed, Lost, MAX_E_ItemHealth);
END_TYPE

(* values of E_PrintSelection: None: Binary Enum. Print A&B = PrintHeadA | PrintHeadB = 0x03 *)

TYPE E_PrintSelection : (None := 16#0, PrintHeadA := 16#1, PrintHeadB := 16#2, MAX_E_PrintSelection);
END_TYPE

(* {attribute 'pack_mode' := '1'} *)
{attribute 'enable_dynamic_creation'}
TYPE T_IdBase_DCH : STRUCT
  rBaseInfo : T_ItemBase;
  udiIdentification : ULINT;  (* Real read process ID values *)
END_STRUCT;
END_TYPE

(* {attribute 'pack_mode' := '1'} *)
{attribute 'enable_dynamic_creation'}
TYPE T_ItemBase : STRUCT
  bolItemAvailable : BOOL;  (* Item Empty *)
  eHealth : E_ItemHealth := E_ItemHealth.Healthy;  (* Actual Status of the item. *)
  uinModuleId : UINT;  (* Actual Position *)
  uinActualPosition : UINT;
  dtStartTimeStamp : TC2_UTILITIES.TIMESTRUCT;
END_STRUCT;
END_TYPE

(* {attribute 'pack_mode' := '1'} *)
{attribute 'enable_dynamic_creation'}
TYPE T_ItemPaperBase : STRUCT
  udiPaperIdProcess : UDINT;  (* Paper ID *)
  udiPaperIdSet : UDINT;  (* Paper ID *)
  bolLastPaperOfStackBatch : UINT;  (* true if this is the paper is the last of a stack. After this paper is placed the stack is ejected. *)
  udiDifferenceToPrevious_ms : UDINT;  (* [ms] Time difference to the previous Paper *)
  udiDifferenceToNext_ms : UDINT;  (* [ms] Time difference to the next paper *)
  eDestination : E_Destination;  (* Paper Stream Destination *)
END_STRUCT;
END_TYPE

TYPE T_GHTHashTableBuffer : STRUCT
  aBuffer : ARRAY[0..(50 - 1)] OF POINTER TO T_HashTableEntry;
END_STRUCT;
END_TYPE

TYPE T_IdBaseRecvData : STRUCT
  fbDataChannel : FB_IdBaseRecvDch;
  rDataChannelItem : T_IdBase_DCH;
  fbFifo : FB_DataChannelRecvFifo;
  rFifoItem : T_IdBase_DCH;
  aFifoBuffer : ARRAY[0..(cRECVDATACHANNELBUFFER - 1)] OF T_IdBase_DCH;
END_STRUCT;
END_TYPE

TYPE T_IdBaseSendData : STRUCT
  fbDataChannel : FB_IdBaseSendDch;
  rDataChannelItem : T_IdBase_DCH;
  fbFifo : FB_DataChannelSenderFifo;
END_STRUCT;
END_TYPE

INTERFACE IBuffer
PROPERTY NumOfItems : DINT
END_PROPERTY
PROPERTY BufferFull : BOOL
END_PROPERTY
PROPERTY MaxCapacity : DINT
END_PROPERTY
END_INTERFACE

INTERFACE IGHT
{attribute 'object_name' := 'AddItem'}
METHOD AddItem : BOOL
  VAR_INPUT
    uliKey : ULINT;
    pData : POINTER TO BYTE;
  END_VAR
END_METHOD
{attribute 'object_name' := 'Lookup'}
METHOD Lookup : POINTER TO BYTE
  VAR_INPUT
    uliKey : ULINT;
    bolRemove : BOOL;
  END_VAR
END_METHOD
{attribute 'object_name' := 'Clear'}
METHOD Clear : BOOL
  VAR_INPUT
    bolFreePointer : BOOL;
  END_VAR
END_METHOD
{attribute 'object_name' := 'Initialize'}
METHOD Initialize : BOOL
END_METHOD
PROPERTY Count : UINT
END_PROPERTY
END_INTERFACE

TYPE U_UMC_Lenze_Control : UNION
  Output : UINT;
  Data : T_UMC_Lenze_Control;
END_UNION;
END_TYPE

TYPE U_UMC_Lenze_Status : UNION
  Input : UINT;
  Data : T_UMC_Lenze_Status;
END_UNION;
END_TYPE

FUNCTION_BLOCK FB_ACL EXTENDS FB_CtrlBase
  VAR
    SIf : T_Ctrl_SIf_ACL;  (* Specific interface struct for public access *)
    fbAddRoute : FB_AddRouteEntry;  (* Used blocks from lib. "utilities" for AMS route handling *)
    fbWrite : ADSWRITE;  (* Used ADS blocks for communication *)
    fbRead : ADSREAD;
    fbReadWrite : ADSRDWRT;
    aListOfConnections : ARRAY[0..cuinMaxConnections] OF T_ADS_ConnectionData;  (* List of all ADS connections handled by this block *)
    uinNumOfAdsConnections : UINT;  (* Number of ADS (server) connections *)
    uinLoopReqHandle : UINT;  (* Loop variable for request of the handle ID *)
    uinConIndex : UINT;  (* Connection index *)
    uinRouteID : UINT;  (* Used for generate unique AMS route names *)
  END_VAR
  VAR CONSTANT
    cSTA_SUB_INITIALIZE : INT := 500;  (* Sub states *)
    cSTA_SUB_READ : INT := 501;
    cSTA_SUB_READBusy : INT := 502;
    cSTA_SUB_WRITE : INT := 503;
    cSTA_SUB_WRITEBusy : INT := 504;
    cSTA_SUB_RW : INT := 505;
    cSTA_SUB_RWBusy : INT := 506;
    cSTA_SUB_ADD_ROUTE : INT := 507;
    cSTA_SUB_ADD_ROUTEBusy : INT := 508;
    cSTA_SUB_ERROR : INT := 509;
    cSTA_SUB_DONE : INT := 510;
    cSTA_SUB_WAIT_NEXT_POLL : INT := 511;
  END_VAR

                  (*__________________________________________________________________________________________________
¦	
¦	Vistaprint Schweiz GmbH
¦	CH - 8401 Winterthur
¦
¦	www.vistaprint.ch - info@vistaprint.ch
¦___________________________________________________________________________________________________

Function desription:
ADS client for data exchange.
Controls the data exchange between various ADS devices. Devices can be added as server connections to that FUB. 

History:
Version		Date			Author		Comment
---------------------------------------------------------------------------------------------------
0.00.1		05.02.2014		AVME/DSC	Start history
0.00.2		17.02.2014		AVME/DSC	BugZilla 140 - Enter ADS route string automatically during state PONBusy

___________________________________________________________________________________________________*)

IF (me.bolActivate) THEN // cyclic call enabled
	IF (CIf.Info.bolInitDone=FALSE) THEN // first cycle -> init
		CtrlInit();
		CIf.Info.bolInitDone := TRUE;
	ELSE
		CycleStartDuty();
	
		Always();
		
		StateMachine();
		
		CycleEndDuty();
	
	END_IF
END_IF;

                

{attribute 'object_name' := 'GetNextAccessType'}
METHOD GetNextAccessType : INT
  VAR_INPUT
    uinNextConnection : UINT;
  END_VAR
                        CASE aListOfConnections[uinNextConnection].eAccessType OF	
	E_ADS_AccessType.READ:
		GetNextAccessType:= cSTA_SUB_READ;	
	E_ADS_AccessType.WRITE:
		GetNextAccessType:= cSTA_SUB_WRITE;	
END_CASE
                      
END_METHOD

{attribute 'object_name' := 'sta_PONBusy'}
METHOD sta_PONBusy : BOOL
  VAR
    stRoute : ST_AmsRouteEntry;
    strRouteName : STRING;
  END_VAR
                        // state implemetation
//--------------------------------------------------------------------------------------
// Entry action
	IF (me.StateMachine.intState<>me.StateMachine.intStateLastCycle) THEN
		me.StateMachine.intStateLastCycle := me.StateMachine.intState;
		
		uinRouteID:= 0;
		uinConIndex:=0;
		// Initialize sub state machine
		me.SubStateMachine.intState:= cSTA_SUB_ADD_ROUTE; 
		me.SubStateMachine.intStateNext := cSTA_SUB_ADD_ROUTE;
		
	END_IF

//--------------------------------------------------------------------------------------
// Cyclic action
	IF (me.StateMachine.intState=me.StateMachine.intStateLastCycle) THEN
		
			// Sub statemachine to set necessary AMS routes and determine the handle ID of all connections in list	
			CASE me.SubStateMachine.intState OF	
			
				// **************************************************************************
				// Call fbAddRoute to add AMS route. Block automatically check if NetID or Name already exist.
				// Double entries not possible!
				// **************************************************************************
				cSTA_SUB_ADD_ROUTE:
				
					// Prepare unique AMS route name: Controller Name: + ID
					uinRouteID:= uinRouteID + 1;
					strRouteName := CONCAT(CIf.Info.strName, ': ID');
					strRouteName := CONCAT(strRouteName, UINT_TO_STRING(uinRouteID));
							
					// Prepare route data
					stRoute.sName:= strRouteName;
					stRoute.sNetID:= aListOfConnections[uinConIndex].strNetID;
					stRoute.sAddress:= THIS^.NetIDtoAddress(aListOfConnections[uinConIndex].strNetID);
					stRoute.eTransport:= eRouteTransport_TCP_IP;
				
					// Add route
					fbAddRoute(bExecute	:= FALSE);
					fbAddRoute( sNetID 	:= '',
								stRoute	:= stRoute,
								bExecute:= TRUE,
								tTimeout:= UDINT_TO_TIME(SIf.Par.udiTOAddRoute_ms),
								bBusy	=>,
								bError	=>,
								nErrID	=>);
				
					me.SubStateMachine.intStateNext := cSTA_SUB_ADD_ROUTEBusy;		
							
				// **************************************************************************
				// Add route busy
				// **************************************************************************
				cSTA_SUB_ADD_ROUTEBusy:
				
					fbAddRoute(bExecute:= FALSE);
					// Add route done
					IF NOT (fbAddRoute.bBusy) THEN
						IF NOT (fbAddRoute.bError) THEN
							// More connections?
							IF (uinConIndex < (uinNumOfAdsConnections-1)) THEN
								uinConIndex:= uinConIndex+1;
								me.SubStateMachine.intStateNext := cSTA_SUB_ADD_ROUTE;
							// All routes added - go on with determine the handle ID 
							ELSE
								uinConIndex:=0;
								me.SubStateMachine.intStateNext := cSTA_SUB_RW;	
							END_IF
						// Error
						ELSE
							// SIf.Alm[7].strText :=  'Adding AMS route failed. Note add. info for affected connection ID';
							pfbAlarmCtrl^.setAlarm(CIf.Info.intCtrlId,7,UDINT_TO_DINT(aListOfConnections[uinConIndex].udiConID),ADR(SIf.Alm),E_AlmState.RST,CIf.Job.eMe_ActivAlmClass);
							me.SubStateMachine.intStateNext := cSTA_SUB_ERROR;		
						END_IF
					END_IF
			
				// **************************************************************************
				// Call fbReadWrite to determine the handle ID
				// **************************************************************************
				cSTA_SUB_RW:
			
					fbReadWrite(WRTRD:= FALSE);
    				fbReadWrite(NETID		:= aListOfConnections[uinConIndex].strNetID,
                				PORT		:= aListOfConnections[uinConIndex].uinTargetPort,
                   				IDXGRP		:= cGET_SYMHANDLE_BYNAME,  
                   				IDXOFFS     := 16#0000,
                   				WRITELEN    := INT_TO_UDINT(LEN(aListOfConnections[uinConIndex].strRoute)+1),
								READLEN     := SIZEOF(aListOfConnections[uinConIndex].udiHandle),
								SRCADDR     := ADR(aListOfConnections[uinConIndex].strRoute),
								DESTADDR    := ADR(aListOfConnections[uinConIndex].udiHandle),
								WRTRD       := TRUE,
								TMOUT       := UDINT_TO_TIME(SIf.Par.udiTORWData_ms),
								BUSY        => ,
								ERR         => ,
								ERRID       => );
								
					me.SubStateMachine.intStateNext := cSTA_SUB_RWBusy;		
				
				// **************************************************************************
				// Read/Write busy
				// **************************************************************************
				cSTA_SUB_RWBusy:
					fbReadWrite(WRTRD:= FALSE);
					// Read/Write done
					IF NOT (fbReadWrite.BUSY) THEN
						IF NOT (fbReadWrite.ERR) THEN
							// More connections?
							IF (uinConIndex < (uinNumOfAdsConnections-1)) THEN
								uinConIndex:= uinConIndex+1;
								me.SubStateMachine.intStateNext := cSTA_SUB_RW;
							// Done - all connection handles are determined 
							ELSE
								me.SubStateMachine.intStateNext := cSTA_SUB_DONE;	
							END_IF
						// Error
						ELSE
							// SIf.Alm[3].strText := 'Init of ADS connection failed. Check add. info for affected connection ID';
							pfbAlarmCtrl^.setAlarm(CIf.Info.intCtrlId,3,UDINT_TO_DINT(aListOfConnections[uinConIndex].udiConID),ADR(SIf.Alm),E_AlmState.RST,CIf.Job.eMe_ActivAlmClass);
							me.SubStateMachine.intStateNext := cSTA_SUB_ERROR;		
						END_IF
					END_IF
				
				// **************************************************************************
				// All necessary AMS routes set and connection handles are determined 
				// **************************************************************************
				cSTA_SUB_DONE:
				
				// **************************************************************************
				// Error
				// **************************************************************************
				cSTA_SUB_ERROR:
				
			END_CASE	
			
		
		// State Change Condition
		IF ((me.SubStateMachine.intState=cSTA_SUB_ERROR) OR (me.StateMachine.udiTimeInState_ms >= SIf.Par.udiTOPowerOn_ms)) THEN
			// In case if TO
			IF (me.StateMachine.udiTimeInState_ms >= SIf.Par.udiTOPowerOn_ms) THEN
				// SIf.Alm[2].strText := 'Timeout initialize ADS connection(s)';
				pfbAlarmCtrl^.setAlarm(CIf.Info.intCtrlId,2,UDINT_TO_DINT(me.StateMachine.udiTimeInState_ms),ADR(SIf.Alm),E_AlmState.RST,CIf.Job.eMe_ActivAlmClass);
			END_IF
			me.StateMachine.intStateNext := cSTA_ERROR;				
		ELSIF (me.SubStateMachine.intState=cSTA_SUB_DONE) THEN
			me.StateMachine.intStateNext := cSTA_PON;
		END_IF
			
	END_IF

//--------------------------------------------------------------------------------------
// Exit action
	IF (me.StateMachine.intState<>me.StateMachine.intStateNext) THEN
		;
	END_IF
                      
END_METHOD

{attribute 'object_name' := 'sta_RUNBusy'}
METHOD sta_RUNBusy : BOOL
                        // state implemetation
//--------------------------------------------------------------------------------------
// Entry action
	IF (me.StateMachine.intState<>me.StateMachine.intStateLastCycle) THEN
		me.StateMachine.intStateLastCycle := me.StateMachine.intState;
		;
	END_IF

//--------------------------------------------------------------------------------------
// Cyclic action
	IF (me.StateMachine.intState=me.StateMachine.intStateLastCycle) THEN
		IF (TRUE) THEN
			me.StateMachine.intStateNext := BASE_PLC.cSTA_RUN;
		END_IF
	END_IF

//--------------------------------------------------------------------------------------
// Exit action
	IF (me.StateMachine.intState<>me.StateMachine.intStateNext) THEN
		;
	END_IF
                      
END_METHOD

{attribute 'object_name' := 'sta_RUN'}
METHOD sta_RUN : BOOL
                        // state implemetation
//--------------------------------------------------------------------------------------
// Entry action
	IF (me.StateMachine.intState<>me.StateMachine.intStateLastCycle) THEN
		me.StateMachine.intStateLastCycle := me.StateMachine.intState;
					
		uinConIndex:=0;
		// Initialize sub state machine
		me.SubStateMachine.intState:= cSTA_SUB_INITIALIZE; 
		me.SubStateMachine.intStateNext := cSTA_SUB_INITIALIZE;
	END_IF

//--------------------------------------------------------------------------------------
// Cyclic action
	IF (me.StateMachine.intState=me.StateMachine.intStateLastCycle) THEN

		// Sub statemachine to handle all connections in list dependent access type (read, write, rw)
		CASE me.SubStateMachine.intState OF	
	
			//************************************************************************
			// Initialize
			//************************************************************************
			cSTA_SUB_INITIALIZE:
				// Get access type
				me.SubStateMachine.intStateNext:= THIS^.GetNextAccessType(uinConIndex);
							
			//************************************************************************					
			// Call fbRead
			//************************************************************************
			cSTA_SUB_READ:
		
				fbRead(READ:= FALSE);
				fbRead(NETID       := aListOfConnections[uinConIndex].strNetID,
						PORT       := aListOfConnections[uinConIndex].uinTargetPort,
						IDXGRP     := cREAD_WRITE_SYMVAL_BYHANDLE,
						IDXOFFS    := aListOfConnections[uinConIndex].udiHandle,
						LEN        := aListOfConnections[uinConIndex].udiDataLen,
						DESTADDR   := aListOfConnections[uinConIndex].pData,
						READ       := TRUE,
						TMOUT      := UDINT_TO_TIME(SIf.Par.udiTOReadData_ms),
						BUSY       => ,
						ERR        => ,
						ERRID      => );
														
				me.SubStateMachine.intStateNext := cSTA_SUB_READBusy;			
							
			//************************************************************************
			// Read busy
			//************************************************************************
			cSTA_SUB_READBusy:
				fbRead(READ:= FALSE);
				// Read done
				IF NOT (fbRead.BUSY) THEN
					IF NOT (fbRead.ERR) THEN	
						// More connections?
						IF (uinConIndex < (uinNumOfAdsConnections-1)) THEN
							uinConIndex:= uinConIndex+1;
							// Get next access type
							me.SubStateMachine.intStateNext:= THIS^.GetNextAccessType(uinConIndex);
						// Done - all connection handles are determined 
						ELSE
							me.SubStateMachine.intStateNext := cSTA_SUB_WAIT_NEXT_POLL;	
						END_IF						
					// Error
					ELSE
						// SIf.Alm[4].strText := 'ADS read data failed. Note add. info to get ADS error ID';
						pfbAlarmCtrl^.setAlarm(CIf.Info.intCtrlId,4,UDINT_TO_DINT(fbRead.ERRID),ADR(SIf.Alm),E_AlmState.RST,CIf.Job.eMe_ActivAlmClass);
						me.SubStateMachine.intStateNext := cSTA_SUB_ERROR;		
					END_IF
				END_IF	
				
			//************************************************************************					
			// Call fbWrite
			//************************************************************************
			cSTA_SUB_WRITE:
		
				fbWrite(WRITE:= FALSE);
				fbWrite(NETID      := aListOfConnections[uinConIndex].strNetID,
						PORT       := aListOfConnections[uinConIndex].uinTargetPort,
						IDXGRP     := cREAD_WRITE_SYMVAL_BYHANDLE,
						IDXOFFS    := aListOfConnections[uinConIndex].udiHandle,
						LEN        := aListOfConnections[uinConIndex].udiDataLen,
						SRCADDR    := aListOfConnections[uinConIndex].pData,
						WRITE      := TRUE,
						TMOUT      := UDINT_TO_TIME(SIf.Par.udiTOWriteData_ms),
						BUSY       => ,
						ERR        => ,
						ERRID      => );
														
				me.SubStateMachine.intStateNext := cSTA_SUB_WRITEBusy;		
				
			//************************************************************************
			// Write busy
			//************************************************************************
			cSTA_SUB_WRITEBusy:
				fbWrite(WRITE:= FALSE);
				// Write done
				IF NOT (fbWrite.BUSY) THEN
					IF NOT (fbWrite.ERR) THEN
						// More connections?
						IF (uinConIndex < (uinNumOfAdsConnections-1)) THEN
							uinConIndex:= uinConIndex+1;
							// Get next access type
							me.SubStateMachine.intStateNext:= THIS^.GetNextAccessType(uinConIndex);
						// Done - all connection handles are determined 
						ELSE
							me.SubStateMachine.intStateNext := cSTA_SUB_WAIT_NEXT_POLL;	
						END_IF
					// Error
					ELSE
						// SIf.Alm[5].strText := 'ADS write data failed. Note add. info to get ADS error ID';
						pfbAlarmCtrl^.setAlarm(CIf.Info.intCtrlId,5,UDINT_TO_DINT(fbWrite.ERRID),ADR(SIf.Alm),E_AlmState.RST,CIf.Job.eMe_ActivAlmClass);
						me.SubStateMachine.intStateNext := cSTA_SUB_ERROR;		
					END_IF
				END_IF			
		
			//************************************************************************
			// Wait for next polling - Connection list completely processed 
			//************************************************************************	
			cSTA_SUB_WAIT_NEXT_POLL:
			
				// Wait polling time expired 	
				IF (me.SubStateMachine.udiTimeInState_ms >= SIf.Par.udiPollingInterval_ms) THEN				
					//Start again at first connection in list
					uinConIndex:=0;
					me.SubStateMachine.intStateNext := cSTA_SUB_INITIALIZE;
				END_IF
				
			//************************************************************************
			// ERROR			
			//************************************************************************	
			cSTA_SUB_ERROR:
				// SIf.Alm[6].strText := 'ADS connection fault. Note add. info for affected connection ID';
				pfbAlarmCtrl^.setAlarm(CIf.Info.intCtrlId,6,UDINT_TO_DINT(aListOfConnections[uinConIndex].udiConID),ADR(SIf.Alm),E_AlmState.RST,CIf.Job.eMe_ActivAlmClass);
				me.StateMachine.intStateNext := BASE_PLC.cSTA_ERROR;	
			
		END_CASE			
	END_IF

//--------------------------------------------------------------------------------------
// Exit action
	IF (me.StateMachine.intState<>me.StateMachine.intStateNext) THEN
		;
	END_IF
                      
END_METHOD

{attribute 'object_name' := 'AddConnection'}
METHOD AddConnection
  VAR_INPUT
    stConnection : T_ADS_ConnectionData;
  END_VAR
                        // Method adds a connection to the internal list of all ADS connections handled by this block
IF (uinNumOfAdsConnections <= (cuinMaxConnections-1)) THEN
	// Add connection to list
	aListOfConnections[uinNumOfAdsConnections] := stConnection;
	// Assigned connection ID
	aListOfConnections[uinNumOfAdsConnections].udiConID := uinNumOfAdsConnections+1;
	// Inc. number of connections
	uinNumOfAdsConnections:= uinNumOfAdsConnections+1;
END_IF
                      
END_METHOD

{attribute 'object_name' := 'StateMachine'}
METHOD StateMachine : BOOL
                        SUPER^.StateMachine();

// main statemachine of base controller
CASE me.StateMachine.intState OF
	cSTA_RUNBusy: 
        THIS^.sta_RUNBusy();
    cSTA_RUN: 
        THIS^.sta_RUN();				
END_CASE;
                      
END_METHOD

{attribute 'object_name' := 'getCmdState'}
METHOD getCmdState : STRING
  VAR_INPUT
    intCmdState : INT;
    bolState : BOOL;
  END_VAR
                        getCmdState := SUPER^.getCmdState(intCmdState:=intCmdState,bolState:=bolState); // get global/base defined cmds/states
IF (getCmdState='') THEN // global not defined get local
	// get string cmd/state string information in runtime
	IF (bolState=FALSE) THEN
		(*
		// cmd's
		CASE intCmdState OF
			;
		END_CASE
		*)
	ELSE
		// states
		CASE intCmdState OF
			// SUB States
			cSTA_SUB_INITIALIZE:
				getCmdState := 'cSTA_SUB_INITIALIZE';
			cSTA_SUB_READ:
				getCmdState := 'cSTA_SUB_READ';
			cSTA_SUB_READBusy:
				getCmdState := 'cSTA_SUB_READBusy';
			cSTA_SUB_WRITE:
				getCmdState := 'cSTA_SUB_WRITE';
			cSTA_SUB_WRITEBusy:
				getCmdState := 'cSTA_SUB_WRITEBusy';			
			cSTA_SUB_RW:
				getCmdState := 'cSTA_SUB_RW';
			cSTA_SUB_RWBusy:
				getCmdState := 'cSTA_SUB_RWBusy';	
			cSTA_SUB_ADD_ROUTE:
				getCmdState := 'cSTA_SUB_ADD_ROUTE';	
			cSTA_SUB_ADD_ROUTEBusy:
				getCmdState := 'cSTA_SUB_ADD_ROUTEBusy';			
			cSTA_SUB_ERROR:
				getCmdState := 'cSTA_SUB_ERROR';
			cSTA_SUB_DONE:
				getCmdState := 'cSTA_SUB_DONE';
			cSTA_SUB_WAIT_NEXT_POLL:
				getCmdState := 'cSTA_SUB_WAIT_NEXT_POLL';
		END_CASE
	END_IF
END_IF
                      
END_METHOD

{attribute 'object_name' := 'getCtrlSIf'}
METHOD getCtrlSIf : POINTER TO T_Ctrl_SIf_ACL
                        getCtrlSIf := ADR(SIf);
                      
END_METHOD

{attribute 'object_name' := 'sta_OFF'}
METHOD sta_OFF : BOOL
                        // state implemetation
//--------------------------------------------------------------------------------------
// Entry action
	IF (me.StateMachine.intState<>me.StateMachine.intStateLastCycle) THEN
		me.StateMachine.intStateLastCycle := me.StateMachine.intState;
		// Initialize sub state machine
		me.SubStateMachine.intState:= cSTA_SUB_INITIALIZE; 
		me.SubStateMachine.intStateNext := cSTA_SUB_INITIALIZE;
	END_IF
	
//--------------------------------------------------------------------------------------
// Cyclic action
	IF (me.StateMachine.intState=me.StateMachine.intStateLastCycle) THEN	
		// State Change Condition
		IF (me.Alarm.eActivAlmClass<>E_AlmClass.EOFF) AND (me.Alarm.eActivAlmClass<>E_AlmClass.OFF) THEN	
			IF(me.intCmd=BASE_PLC.cCMD_RUN) THEN
				me.StateMachine.intStateNext := BASE_PLC.cSTA_RUNBusy;
			END_IF
		END_IF
	END_IF

//--------------------------------------------------------------------------------------
// Exit action
	IF (me.StateMachine.intState<>me.StateMachine.intStateNext) THEN
		;
	END_IF
                      
END_METHOD

{attribute 'object_name' := 'Always'}
METHOD Always : BOOL
                        SUPER^.Always();

// ----------------------------------------------------------------------------------
// cyclic actions outside of statemachine
IF (me.StateMachine.intState<>cSTA_SINGLE_ANSWER) THEN
	SIf.Cur.uinNumOfAdsConnections:= uinNumOfAdsConnections;	
END_IF

// If no connection added, set alarm and change to state error
IF (uinNumOfAdsConnections = 0) THEN
	// Set Alarm: SIf.Alm[1].strText := 'Initialization error. Minimum one ADS connection must be configured'; 
	pfbAlarmCtrl^.setAlarm(CIf.Info.intCtrlId,1,0,ADR(SIf.Alm),E_AlmState.RST,CIf.Job.eMe_ActivAlmClass);	
	me.StateMachine.intStateNext := BASE_PLC.cSTA_ERROR;
END_IF

// ----------------------------------------------------------------------------------
// Always change actions in Base Library
// ----------------------------------------------------------------------------------
// overrule error always from base -> no EOFF State!! in EOFF go to OFF
IF (me.StateMachine.intStateNext = cSTA_EOFFBusy) THEN
	IF (me.StateMachine.intState=cSTA_OFF) THEN
		me.StateMachine.intStateNext := cSTA_OFF;
	ELSE // stay in OFF
		me.StateMachine.intStateNext := cSTA_OFFBusy;
	END_IF
END_IF
                      
END_METHOD

{attribute 'object_name' := 'sta_PON'}
METHOD sta_PON : BOOL
                        // state implemetation
//--------------------------------------------------------------------------------------
// Entry action
	IF (me.StateMachine.intState<>me.StateMachine.intStateLastCycle) THEN
		me.StateMachine.intStateLastCycle := me.StateMachine.intState;
		
	END_IF

//--------------------------------------------------------------------------------------
// Cyclic action
	IF (me.StateMachine.intState=me.StateMachine.intStateLastCycle) THEN
		
		;	
		// State Change Condition
		IF (me.intCmd<>cCMD_PON) AND (me.intCmd<>cCMD_DONE) THEN
			me.StateMachine.intStateNext := BASE_PLC.cSTA_OFFBusy;
		END_IF
	END_IF

//--------------------------------------------------------------------------------------
// Exit action
	IF (me.StateMachine.intState<>me.StateMachine.intStateNext) THEN
		;
	END_IF
                      
END_METHOD

{attribute 'object_name' := 'NetIDtoAddress'}
METHOD NetIDtoAddress : STRING
  VAR_INPUT
    strNetID : STRING;
  END_VAR
  VAR
    intI : INT;
    strCharacter : STRING(1);
    uinExitCounter : UINT;
    cDot : USINT := 16#2E;
  END_VAR
                        // Method convert a ADS NetID to a standard IP Address
// Example: 192.168.70.27.1.1 -> 192.168.70.27
uinExitCounter:=0;
// Get all numbers up to 4 point
FOR intI:=0 TO LEN(strNetID) DO	
	// Get single char
	strCharacter:= Mid(strNetID,1,intI);
	// Incr. exit counter if char = '.'
	IF (F_ToASC(strCharacter) = cDot) THEN
		uinExitCounter:= uinExitCounter +1;
	END_IF
	// As long as 4 point not reached
	IF uinExitCounter < 4 THEN
		NetIDtoAddress:= CONCAT(NetIDtoAddress,strCharacter);	
	ELSE
		EXIT;
	END_IF 
END_FOR





                      
END_METHOD

{attribute 'object_name' := 'FB_init'}
METHOD FB_init : BOOL
  VAR_INPUT
    bInitRetains : BOOL;  (* if TRUE, the retain variables are initialized (warm start / cold start) *)
    bInCopyCode : BOOL;  (* if TRUE, the instance afterwards gets moved into the copy code (online change) *)
  END_VAR
  VAR
    udiTaskCnt : UDINT;
    ii : UINT;
  END_VAR
                        //------------------------------------------------------------------------------------------------------------------------
// to manually change in new FUB implementation!!!
// define valid commands for this controller
FOR ii:= 0 TO (SIZEOF(CIf.Job.aCmdList)/SIZEOF(CIf.Job.aCmdList[0])-1) BY 1 DO
	IF (CIf.Job.aCmdList[ii].intCmd=cCMD_INITIALIZED) THEN
		// found first empty array element
		EXIT;
	END_IF
END_FOR
CIf.Job.aCmdList[ii].intCmd := cCMD_RUN;
CIf.Job.aCmdList[ii].strName := 'Run'; 
CIf.Job.aCmdList[ii].bolAvailable := TRUE;
ii := ii +1;

// set name of class/typ
CIf.Info.strType := 'FB_ACL';
CIf.Info.strFullName := 'ADS Client';

// set alarm class
SIf.Alm[1].eAlmClass := E_AlmClass.OFF;
SIf.Alm[1].strText := 'Initialization error. Minimum one ADS connection must be configured'; 
SIf.Alm[2].eAlmClass := E_AlmClass.OFF;
SIf.Alm[2].strText := 'Timeout initialize ADS connection(s)';
SIf.Alm[3].eAlmClass := E_AlmClass.OFF;
SIf.Alm[3].strText := 'Init of ADS connection failed. Note add. info for affected connection ID';
SIf.Alm[4].eAlmClass := E_AlmClass.OFF;
SIf.Alm[4].strText := 'ADS read data failed. Note add. info to get ADS error ID';
SIf.Alm[5].eAlmClass := E_AlmClass.OFF;
SIf.Alm[5].strText := 'ADS write data failed. Note add. info to get ADS error ID';
SIf.Alm[6].eAlmClass := E_AlmClass.OFF;
SIf.Alm[6].strText := 'ADS connection fault. Note add. info for affected connection ID';
SIf.Alm[7].eAlmClass := E_AlmClass.OFF;
SIf.Alm[7].strText :=  'Adding AMS route failed. Note add. info for affected connection ID';

//*******************************************************************************
// initial values
//*******************************************************************************

// software configuration
CIf.SwCfg.bolExist := TRUE;
CIf.SwCfg.bolSimulation := FALSE;

// parameter
SIf.Par.udiTOAddRoute_ms:= 1500;
SIf.Par.udiTOPowerOn_ms:= 10000;
SIf.Par.udiTOReadData_ms:= 1500;
SIf.Par.udiTOWriteData_ms:= 1500;
SIf.Par.udiTORWData_ms:= 1500;
SIf.Par.udiPollingInterval_ms:= 100;
                      
END_METHOD

{attribute 'object_name' := 'sta_ERROR'}
METHOD sta_ERROR : BOOL
                        // state implemetation
//--------------------------------------------------------------------------------------
// Entry action
	IF (me.StateMachine.intState<>me.StateMachine.intStateLastCycle) THEN
		me.StateMachine.intStateHistory := me.StateMachine.intStateLastCycle; // -> possibillity to go back to state before error
		me.StateMachine.intStateLastCycle := me.StateMachine.intState;
		
		// Initialize sub state machine
		me.SubStateMachine.intState:= cSTA_SUB_INITIALIZE; 
		me.SubStateMachine.intStateNext := cSTA_SUB_INITIALIZE;
	END_IF

//--------------------------------------------------------------------------------------
// Cyclic action
	IF (me.StateMachine.intState=me.StateMachine.intStateLastCycle) THEN
		// State Change Condition
		IF (CIf.Job.bolAlmReset = TRUE) THEN
			me.StateMachine.intStateNext := cSTA_ERRORQuit;
		END_IF
	END_IF

//--------------------------------------------------------------------------------------
// Exit action
	IF (me.StateMachine.intState<>me.StateMachine.intStateNext) THEN
		;
	END_IF
                      
END_METHOD

PROPERTY CtrlSIf : POINTER TO T_Ctrl_SIf_ACL
GET
                          CtrlSIf := ADR(SIf);
                        
END_GET
END_PROPERTY
END_FUNCTION_BLOCK

FUNCTION_BLOCK FB_BCD
  VAR
    bolInitDone : BOOL;
    bolActivate : BOOL := TRUE;
    SIf : T_BCD;  (* driver specific interface *)
    stStateMachine : T_BCD_StateMachine;
    stSubStateMachine : T_BCD_StateMachine;
    fbClientConnection : FB_ClientServerConnection;  (* Create/release TCP/IP connection *)
    fbSend : FB_SocketSend;  (* Send TCP/IP data *)
    fbReceive : FB_SocketReceive;  (* Receive TCP/IP data *)
    aRxData : ARRAY[0..300] OF BYTE;  (* Rx data buffer *)
    rTxData : T_BCD_TxStructure;  (* Tx data *)
    intTxState : INT;
    bolExecuteSend : BOOL;
    udiNSend : UDINT;  (* counter for sended frames *)
    intRxState : INT;
    bolExecuteRead : BOOL;
    udiReceivedBytes : UDINT;  (* Count of received data bytes *)
    strReceivedMessage : STRING(255);
    iStringLength : INT;
    iReaderType : E_BCD_Type;  (* bar code reader type *)
  END_VAR
  VAR CONSTANT
    cBCD_SUB_Send : INT := 2000;
    cBCD_SUB_Wait : INT := 2001;
    cBCD_SUB_Read : INT := 2002;
    cBCD_SUB_CheckAnswer : INT := 2003;
    cBCD_SUB_GetData : INT := 2004;
    cBCD_SUB_Done : INT := 2005;
    cBCD_SUB_Error : INT := 2006;
    cTxIdle : USINT := 0;
    cTxBusy : USINT := 1;
    cRxIdle : USINT := 0;
    cRxBusy : USINT := 1;
    cRxConv : USINT := 2;
    cSTX : USINT := 16#2;
    cETX : USINT := 16#3;
    cCR : USINT := 16#D;
    cLF : USINT := 16#A;
  END_VAR

                  (*__________________________________________________________________________________________________
¦	
¦	Vistaprint Schweiz GmbH
¦	CH - 8401 Winterthur
¦
¦	www.vistaprint.ch - info@vistaprint.ch
¦___________________________________________________________________________________________________

Function desription:
TCP-IP driver for SICK barcode reader CLV632-0120
Note: This driver work as a TCP client.

History:
Version		Date			Author		Comment
---------------------------------------------------------------------------------------------------
0.00.1		18.12.2013		AVME/DSC	Start history
0.00.2		03.01.2014		AVME/DSC	Basic functionalities implemented and tested. Following commands are supported:
										CMD_CONNECT_SOCKET 	1002 		// Connect TCP socket
										CMD_CLOSE_SOCKET 	1004 		// Close TCP socket
										CMD_COM_TEST 		1006 		// Communication test 
										CMD_READ_BARCODE 	1014 		// Command enable the sensor gate for X-TIME ("duration" setting of sensor object trigger)
																		// Sensor try to detect a barcode.
0.00.3		27.01.2014		AVME/DSC    Added new method "CheckSensorError" to set "bolSensorError" in case if sensor answer with SOPAS error																					 							
0.00.4		24.10.2014		HLV/MAH		driver can be used for Sick or Keyence scanner configured by SIf.Cfg.iSensorType := E_BCD_Type.xxxx
										the port of Keyence scanner must be always 9004
										if Keyence scanner is used, FB_SocketCloseAll must be called in main PRG (see MiddlePRG in BaseElementsSample)

	
___________________________________________________________________________________________________*)


IF (bolActivate) THEN // cyclic call enabled
	
	IF (bolInitDone=FALSE) THEN // first cycle -> init
		CtrlInit();	
		bolInitDone := TRUE;
	ELSE
		CycleStartDuty();
				
		StateMachine();
		
		CycleEndDuty();
	END_IF
	
END_IF;
                

ACTION ClearTxBuffer:
                      Tc2_System.MEMSET(ADR(rTxData.aTxData),16#00,SIZEOF(rTxData.aTxData));

                    
END_ACTION

{attribute 'object_name' := 'sta_ConnectSocketBusy'}
METHOD sta_ConnectSocketBusy : BOOL
                        // state implemetation
//--------------------------------------------------------------------------------------
// Entry action
	IF (stStateMachine.intState<>stStateMachine.intStateLastCycle) THEN
		stStateMachine.intStateHistory := stStateMachine.intStateLastCycle;
		stStateMachine.intStateLastCycle := stStateMachine.intState;
			
		// Initialize and connect socket
		fbClientConnection.nMode := CONNECT_MODE_ENABLEDBG; 			// not used
		fbClientConnection.sRemoteHost := SIf.stCfg.strSensorIPAdr;
		fbClientConnection.nRemotePort := SIf.stCfg.udiSensorPort;
		fbClientConnection.tReconnect := SIf.stPar.tTOConnection;
		fbClientConnection.bEnable:= TRUE;

	END_IF

//--------------------------------------------------------------------------------------
// Cyclic action
	IF (stStateMachine.intState=stStateMachine.intStateLastCycle) THEN
		
	
		// State Change Condition

		// Check about FUB error	
		IF (fbClientConnection.bError = TRUE) OR (fbClientConnection.nErrId <> 0) THEN
			SIf.stErr.bolErrorActive := TRUE;	
			SIf.stErr.bolSocketError := TRUE;
			SIf.stErr.udiErrorID := fbClientConnection.nErrId;
			stStateMachine.intStateNext := cBCD_STA_Error;
		END_IF
	
		// Wait for socket handle ID	
		IF (fbClientConnection.hSocket.handle <> 0) AND (fbClientConnection.eState = eSOCKET_CONNECTED) THEN
			stStateMachine.intStateNext := cBCD_STA_WaitForJob;
		END_IF

	END_IF

//--------------------------------------------------------------------------------------
// Exit action
	IF (stStateMachine.intState<>stStateMachine.intStateNext) THEN
		SIf.intCmd := cBCD_CMD_DONE;
	END_IF
                      
END_METHOD

{attribute 'object_name' := 'CycleStartDuty'}
METHOD CycleStartDuty : BOOL
                        // ----------------------------------------------------------------------------------
// cyclic actions outside of statemachine

// Simulation active
IF (SIf.stCfg.bolSimulation) THEN
	;
ELSE
	;
END_IF

// Cyclic call of the client connection
fbClientConnection();
// Cyclic call of method "HandleRxData"
THIS^.HandleRxData();

// Generate socket connected status info
IF (fbClientConnection.eState = eSOCKET_CONNECTED) THEN
	SIf.stStatus.bolSocketConnected:= TRUE;
ELSE
	SIf.stStatus.bolSocketConnected:= FALSE;	
	SIf.stStatus.bolComChecked:= FALSE;
END_IF

// Command close socket can be executed all the time.
// Used for error recovery in case if parent controller has an error.
IF (SIf.intCmd=cBCD_CMD_CLOSE_SOCKET) THEN	
	stStateMachine.intStateNext := cBCD_STA_CloseSocketBusy;
END_IF
			
SIf.strCmd := THIS^.getCmdState(intCmdState:=SIf.intCmd,bolState:=FALSE);
                      
END_METHOD

{attribute 'object_name' := 'PrepareReadMsg'}
METHOD PrepareReadMsg
  VAR
    uinI : UINT;
    strCharacter : STRING(1);
  END_VAR
                        // Delete last message
strReceivedMessage:= '';

// Loop over receive buffer
FOR uinI:= 0 TO SIZEOF(aRxData)-1 DO	
	// Start of text?
	IF (aRxData[uinI] = cSTX) THEN
		;
	// End of text?
	ELSIF (aRxData[uinI] = cETX) THEN
		EXIT;
	ELSE
		// Convert ASCII to string
		strCharacter:= F_ToCHR(aRxData[uinI]);
		strReceivedMessage:= CONCAT(strReceivedMessage,strCharacter);			
	END_IF
END_FOR
                      
END_METHOD

{attribute 'object_name' := 'sta_SocketClosed'}
METHOD sta_SocketClosed : BOOL
                        // state implemetation
//--------------------------------------------------------------------------------------
// Entry action
	IF (stStateMachine.intState<>stStateMachine.intStateLastCycle) THEN
		stStateMachine.intStateLastCycle := stStateMachine.intState;
		;
	END_IF

//--------------------------------------------------------------------------------------
// Cyclic action
	IF (stStateMachine.intState=stStateMachine.intStateLastCycle) THEN

		// State Change Condition
		IF (SIf.intCmd=cBCD_CMD_CONNECT_SOCKET) THEN
			stStateMachine.intStateNext := cBCD_STA_ConnectSocketBusy;
		END_IF
		
	END_IF

//--------------------------------------------------------------------------------------
// Exit action
	IF (stStateMachine.intState<>stStateMachine.intStateNext) THEN
		;
	END_IF
                      
END_METHOD

{attribute 'object_name' := 'sta_CloseSocketBusy'}
METHOD sta_CloseSocketBusy : BOOL
                        // state implemetation
//--------------------------------------------------------------------------------------
// Entry action
	IF (stStateMachine.intState<>stStateMachine.intStateLastCycle) THEN
		stStateMachine.intStateHistory := stStateMachine.intStateLastCycle;
		stStateMachine.intStateLastCycle := stStateMachine.intState;
		
		// Reset pending commands			
		bolExecuteSend:= FALSE;
		bolExecuteRead:= FALSE;
		// Reset Rx/Tx states
		intRxState:= cRxIdle;
		intTxState:= cTxIdle;
		// Close socket
		fbClientConnection.bEnable:= FALSE;

	END_IF

//--------------------------------------------------------------------------------------
// Cyclic action
	IF (stStateMachine.intState=stStateMachine.intStateLastCycle) THEN
		
	
		// State Change Condition

		// Check about FUB error	
		IF (fbClientConnection.bError = TRUE) OR (fbClientConnection.nErrId <> 0) THEN
			SIf.stErr.bolErrorActive := TRUE;	
			SIf.stErr.bolSocketError := TRUE;
			SIf.stErr.udiErrorID := fbClientConnection.nErrId;
			stStateMachine.intStateNext := cBCD_STA_Error;
		END_IF
	
		// Wait until socket is closed	
		IF (fbClientConnection.eState = eSOCKET_CLOSED) THEN
			stStateMachine.intStateNext := cBCD_STA_WaitForJob;
		ELSIF  (SIf.stErr.bolErrorActive= TRUE) THEN 
			stStateMachine.intStateNext := cBCD_STA_Error;		
		END_IF
	
	END_IF

//--------------------------------------------------------------------------------------
// Exit action
	IF (stStateMachine.intState<>stStateMachine.intStateNext) THEN
		SIf.intCmd := cBCD_CMD_DONE;
	END_IF
                      
END_METHOD

{attribute 'object_name' := 'CycleEndDuty'}
METHOD CycleEndDuty : BOOL
                        SIf.strState := THIS^.getCmdState(intCmdState:=stStateMachine.intState,bolState:=TRUE);

IF (stStateMachine.intState<>stStateMachine.intStateNext) THEN
	stStateMachine.intState := stStateMachine.intStateNext;  // set next state for next cycle
END_IF

(***************************************************************
        Function Block Calls
***************************************************************)

// Cyclic call of method "HandleTxData"
THIS^.HandleTxData();
                      
END_METHOD

{attribute 'object_name' := 'HandleRxData'}
METHOD HandleRxData
  VAR
    uinI : UINT;
  END_VAR
                        // GET/FETCH RX DATA
CASE intRxState OF
	
	// wait for read command
	cRxIdle:
		IF (bolExecuteRead=TRUE) AND (fbClientConnection.eState = eSOCKET_CONNECTED)THEN	

			// clear rx buffer
			FOR uinI:= 0 TO SIZEOF(aRxData)-1 DO
				aRxData[uinI]:= 16#00;
			END_FOR
			// Delete last message
			strReceivedMessage:= '';
			udiReceivedBytes := 0;
								
			// receive frame			
			fbReceive( bExecute := FALSE );
			fbReceive( 	sSrvNetId	:= '',
						hSocket		:= fbClientConnection.hSocket,
						cbLen		:= SIZEOF(aRxData),
						pDest		:= ADR(aRxData),
						bExecute	:= TRUE,
						tTimeout	:= SIf.stPar.tTOReceive);
			intRxState := cRxBusy;		
		END_IF
		
	// wait until receive not busy
	cRxBusy:
		fbReceive( bExecute := FALSE );
		IF NOT fbReceive.bBusy THEN
			IF NOT fbReceive.bError THEN
				IF (fbReceive.nRecBytes > 0) THEN (* some bytes received *)
					udiReceivedBytes := fbReceive.nRecBytes;
					intRxState := cRxConv; // convert received message
				ELSE
					// Try to read again
					intRxState := cRxIdle;
				END_IF	
			// Error	
			ELSE
				IF (SIf.stErr.bolErrorActive = FALSE) THEN
					SIf.stErr.bolErrorActive := TRUE;	
					SIf.stErr.udiErrorID := fbReceive.nErrId;	
					// Try to close the socket. Needs reconnect for socket after an error!	
					stStateMachine.intStateNext := cBCD_STA_CloseSocketBusy;	
				END_IF	
			END_IF			
		END_IF
			
	// convert received message to string
	cRxConv: 
		THIS^.PrepareReadMsg();
		THIS^.CheckSensorError(); // Error response: [STX]sFA <x>[ETX]    	
		bolExecuteRead:= FALSE; // Read done and data converted to string format
		intRxState := cRxIdle;
		
END_CASE

                      
END_METHOD

{attribute 'object_name' := 'sta_Error'}
METHOD sta_Error : BOOL
                        // state implemetation
//--------------------------------------------------------------------------------------
// Entry action
	IF (stStateMachine.intState<>stStateMachine.intStateLastCycle) THEN
		stStateMachine.intStateHistory := stStateMachine.intStateLastCycle;
		stStateMachine.intStateLastCycle := stStateMachine.intState;
		
		// Reset pending commands			
		bolExecuteSend:= FALSE;
		bolExecuteRead:= FALSE;
		// Reset Rx/Tx states
		intRxState:= cRxIdle;
		intTxState:= cTxIdle;
		
	END_IF


//--------------------------------------------------------------------------------------
// Cyclic action
	IF (stStateMachine.intState=stStateMachine.intStateLastCycle) THEN
			
		// State Change Condition
		IF (SIf.stErr.bolErrAck = TRUE) THEN
			// Reset all active errors
			SIf.stErr.bolErrorActive := FALSE;
			SIf.stErr.bolSocketError := FALSE;
			SIf.stErr.bolSensorError := FALSE;
			SIf.stErr.udiErrorID := 0;
			SIf.stErr.bolErrAck := FALSE;
			// Needs reconnect for socket after an error!		
			stStateMachine.intStateNext := cBCD_STA_CloseSocketBusy;		
		END_IF
		
	END_IF

//--------------------------------------------------------------------------------------
// Exit action
	IF (stStateMachine.intState<>stStateMachine.intStateNext) THEN
		;
	END_IF
                      
END_METHOD

{attribute 'object_name' := 'StateMachine'}
METHOD StateMachine : BOOL
                        
// main statemachine
CASE stStateMachine.intState OF	
	cBCD_STA_WaitForJob:
   		THIS^.sta_WaitForJob();
	cBCD_STA_ConnectSocketBusy: 
        THIS^.sta_ConnectSocketBusy();	
	cBCD_STA_CloseSocketBusy: 
        THIS^.sta_CloseSocketBusy();		
	cBCD_STA_SocketClosed: 
        THIS^.sta_SocketClosed();	
	cBCD_STA_ComTestBusy:
	    THIS^.sta_ComTestBusy();
	cBCD_STA_ReadCodeBusy:
	    THIS^.sta_ReadCodeBusy();
    cBCD_STA_Error: 
        THIS^.sta_Error();
END_CASE;
                      
END_METHOD

{attribute 'object_name' := 'getSIf'}
METHOD getSIf : POINTER TO T_BCD
                        getSIf := ADR(SIf);
                      
END_METHOD

{attribute 'object_name' := 'getCmdState'}
METHOD getCmdState : STRING
  VAR_INPUT
    intCmdState : INT;
    bolState : BOOL;
  END_VAR
                        // get string cmd/state string information in runtime
IF (bolState=FALSE) THEN
	
// cmd's
	CASE intCmdState OF
		cBCD_CMD_DONE: 
			getCmdState := 'cBCD_CMD_DONE';
		cBCD_CMD_CONNECT_SOCKET: 
			getCmdState := 'cBCD_CMD_CONNECT_SOCKET';
		cBCD_CMD_CLOSE_SOCKET: 
			getCmdState := 'cBCD_CMD_CLOSE_SOCKET';
		cBCD_CMD_READ_BARCODE: 
			getCmdState := 'cBCD_CMD_READ_BARCODE';		
		cBCD_CMD_COM_TEST: 
			getCmdState := 'cBCD_CMD_COM_TEST';			
	END_CASE;
ELSE

// state's
	CASE intCmdState OF
		cBCD_STA_WaitForJob: 
			getCmdState := 'cBCD_STA_WaitForJob';
		cBCD_STA_ConnectSocketBusy: 
			getCmdState := 'cBCD_STA_ConnectSocketBusy';
		cBCD_STA_CloseSocketBusy: 
			getCmdState := 'cBCD_STA_CloseSocketBusy';
		cBCD_STA_SocketClosed: 
			getCmdState := 'cBCD_STA_SocketClosed';	
		cBCD_STA_ReadCodeBusy: 
			getCmdState := 'cBCD_STA_ReadCodeBusy';	
		cBCD_STA_ComTestBusy:
			getCmdState := 'cBCD_STA_ComTestBusy';	
		cBCD_STA_Error: 
			getCmdState := 'cBCD_STA_Error';
	END_CASE;
	
END_IF


                      
END_METHOD

{attribute 'object_name' := 'HandleTxData'}
METHOD HandleTxData
                        // HANDLE TX DATA
CASE intTxState OF
	
	// wait for send command (ready for send)
	cTxIdle:
		IF (bolExecuteSend) AND (fbClientConnection.eState = eSOCKET_CONNECTED)THEN									
			// send frame
			fbSend( bExecute := FALSE );
			fbSend(	sSrvNetID 	:= '',
					hSocket		:= fbClientConnection.hSocket,
					cbLen		:= rTxData.intMessageSize,
					pSrc		:= ADR(rTxData.aTxData),					// pointer to the frame data
					bExecute	:= TRUE,
					tTimeout 	:= SIf.stPar.tTOSend);
	
			intTxState := cTxBusy;							
		END_IF
		
	// wait until send not busy
	cTxBusy:
		fbSend( bExecute := FALSE );
		IF NOT (fbSend.bBusy) THEN
			intTxState := cTxIdle;
			// Check about FUB error	
			IF (fbSend.bError = TRUE) THEN
				IF (SIf.stErr.bolErrorActive = FALSE) THEN
					SIf.stErr.bolErrorActive := TRUE;	
					SIf.stErr.udiErrorID := fbSend.nErrId;	
					// Try to close the socket. Needs reconnect for socket after an error!	
					stStateMachine.intStateNext := cBCD_STA_CloseSocketBusy;	
				END_IF				
			// no error
			ELSE
				udiNSend := udiNSend + 1; // increment the number of send frames
				bolExecuteSend:= FALSE;
			END_IF
		END_IF
		
END_CASE
                      
END_METHOD

{attribute 'object_name' := 'sta_ComTestBusy'}
METHOD sta_ComTestBusy : BOOL
                        // state implemetation
//--------------------------------------------------------------------------------------
// Entry action
	IF (stStateMachine.intState<>stStateMachine.intStateLastCycle) THEN
		stStateMachine.intStateHistory := stStateMachine.intStateLastCycle;
		stStateMachine.intStateLastCycle := stStateMachine.intState;

		// Clear data
		SIf.stData.stDevInfo.strComTestResult:='';
		SIf.stStatus.bolComChecked:=FALSE;
	
		// Init sub state machine
		stSubStateMachine.intState := cBCD_SUB_Send;
		stSubStateMachine.intStateNext := cBCD_SUB_Send;	
	END_IF

//--------------------------------------------------------------------------------------
// Cyclic action
	IF (stStateMachine.intState=stStateMachine.intStateLastCycle) THEN
			
		// sub state machine for reading the bar code	
		CASE stSubStateMachine.intState OF

			cBCD_SUB_Send:
				// Check Tx state idle
				IF (intTxState = cTxIdle) THEN
					CASE SIf.stCfg.iSensorType OF
						E_BCD_Type.SICK:
							THIS^.PrepareSendMsg('sRI0'); // Call SOPAS command "sRI0"
							
						E_BCD_Type.KEYENCE:
							THIS^.PrepareSendMsg('BCLR'); // clear send buffer
					END_CASE
					bolExecuteSend:= TRUE;
					stSubStateMachine.intState := cBCD_SUB_Wait;
				END_IF
		
			cBCD_SUB_Wait:
				// Wait until executed -> flag set back to false by method handle TxData
				IF (bolExecuteSend=FALSE)THEN
					stSubStateMachine.intState := cBCD_SUB_Read;
				END_IF
				
			cBCD_SUB_Read:
				// Check Rx state idle
				IF (intRxState = cRxIdle) THEN
					bolExecuteRead:= TRUE;
					stSubStateMachine.intState := cBCD_SUB_CheckAnswer;
				END_IF
			
			cBCD_SUB_CheckAnswer:
				// Wait until executed -> flag set back to false by method handle RxData
				IF (bolExecuteRead=FALSE)THEN				
					// Check about corresponding answer for the command	
					CASE SIf.stCfg.iSensorType OF
						E_BCD_Type.SICK:					
							IF (TC2_STANDARD.FIND(strReceivedMessage,'sRA') <> 0) THEN
								SIf.stData.stDevInfo.strComTestResult:=strReceivedMessage;
								SIf.stStatus.bolComChecked:=TRUE;
							END_IF
						
						E_BCD_Type.KEYENCE:
							IF (TC2_STANDARD.FIND(strReceivedMessage,'OK,BCLR') <> 0) THEN
								SIf.stData.stDevInfo.strComTestResult:=strReceivedMessage;
								SIf.stStatus.bolComChecked:=TRUE;
							END_IF
					END_CASE
					stSubStateMachine.intState := cBCD_SUB_Done;
				END_IF
			
			cBCD_SUB_Done:
				; // job executed
			
		END_CASE
		
		 // job executed
		IF (stSubStateMachine.intState = cBCD_SUB_Done) THEN
			stStateMachine.intStateNext := cBCD_STA_WaitForJob;	
		END_IF
	
	END_IF

//--------------------------------------------------------------------------------------
// Exit action
	IF (stStateMachine.intState<>stStateMachine.intStateNext) THEN
		SIf.intCmd := cBCD_CMD_DONE;
	END_IF
                      
END_METHOD

{attribute 'object_name' := 'FB_init'}
METHOD FB_init : BOOL
  VAR_INPUT
    bInitRetains : BOOL;  (* if TRUE, the retain variables are initialized (warm start / cold start) *)
    bInCopyCode : BOOL;  (* if TRUE, the instance afterwards gets moved into the copy code (online change) *)
  END_VAR
                        // Communication Settings
SIf.stCfg.strSensorIPAdr := '192.168.1.103';  //'192.168.0.10'; 
SIf.stCfg.udiSensorPort := 9004;
SIf.stCfg.bolResponseIncludingDiagnostics := FALSE;
SIf.stCfg.iSensorType := E_BCD_Type.KEYENCE;

// Parameter
SIf.stPar.tTOConnection := T#50S;
SIf.stPar.tTOReceive := T#5S;
SIf.stPar.tTOSend := T#5S;
                      
END_METHOD

{attribute 'object_name' := 'PrepareBarCodeData'}
METHOD PrepareBarCodeData
  VAR
    intI : INT;
    intStartIndex : INT;
    intStartIndexCode : INT;
    bASCIISign : BYTE;
    strCharacter : STRING(1);
  END_VAR
                        
// Note: Currently only the bar code is read out from the received message. "OI=" section in message.
// Other data sections like e.g. "TT=", "OTL=", "CC=" are not prepared.

// ----------------------------------------------------
// Get bar code and write result to structure "stData"
// ----------------------------------------------------
	
// Example of message: <stx> <CR><LF> TT=125ms OTL=0mm CC=1 OI=25<CR><LF>45376049874<CR><LF> .... and so on ...   <etx>
				 
// Get start index for bar code 'OI='
intStartIndex := TC2_STANDARD.FIND(strReceivedMessage,'OI=');

// Loop over received message to get the bar code
FOR intI:=intStartIndex TO LEN(strReceivedMessage)-intStartIndex DO	
	// Convert to ASCII to detect CR and LF
	bASCIISign:= F_ToASC(Mid(strReceivedMessage,1,intI));
	// The bar code number starts after LF					
	IF (bASCIISign = cLF) THEN
		// Save start index of the bar code
		intStartIndexCode:= intI + 1;
	END_IF
	// Read every single number of the bar code until the end "CR"
	IF ((intStartIndexCode <> 0) AND (intI >= intStartIndexCode)) THEN
		// As long as the end is not reached...(The bar code number ends with CR)	
		IF (bASCIISign <> cCR) THEN								
			// Write result to structure stData	
			strCharacter:= Mid(strReceivedMessage,1,intI);
			SIf.stData.strBarCode:= CONCAT(SIf.stData.strBarCode,strCharacter);	
			SIf.stData.uliBarCode:= STRING_TO_ULINT(SIf.stData.strBarCode);
			SIf.stData.bolCodeReaded:= TRUE;																	
		ELSE
			// end of bar code reached "CR" -> EXIT loop
			EXIT;
		END_IF
	END_IF
	
END_FOR
                      
END_METHOD

{attribute 'object_name' := 'CheckSensorError'}
METHOD CheckSensorError
  VAR
    strErrorID : STRING(3);
    bytErrorID : BYTE;
    cbData : UDINT;
  END_VAR
                        (*--------------------------------------------------------------------------
IF an error occurs the Sopas command is answered with:
[STX]sFA <x>[ETX] as an error response

	Error list: <x> can have following values:
	1:	Access denied
	2:	Unknown Index
	3:	Unknown Index
	4:	Wrong Condition
	5:	Invalid Data
	6:	Unknown Error
	7:	Too Many Parameter
	8:	Parameter Missing
	9: 	Wrong Parameter
	A:	No Write Access
	B:	Unknown Command
	C:	Unknown Command
	D:	Server Busy
	E:	Textstring Too Long
	F:	Unknown Event
	10:	Too many Parameter
	11: Invalid Character
	12.	No Message
	13:	No Answer
	14:	Internal Error
	15:	HubAddress: wrong
	16:	HubAddress: error
	17:	HubAddress: error

---------------------------------------------------------------------------*)

// If received message is an error response from sensor: [STX]sFA <x>[ETX]    				
IF (TC2_STANDARD.FIND(strReceivedMessage,'sFA') <> 0) THEN
	
	// Get error number
	strErrorID := Mid(strReceivedMessage,LEN(strReceivedMessage)-1,5);
	cbData := HEXSTR_TO_DATA( strErrorID, ADR(bytErrorID), SIZEOF(bytErrorID));

	// No interpretation of the error number, only set SensorError with error number info 
	(*
	CASE bytErrorID OF
		16#1: 
		16#2:
		16#3:	
		16#A:			
		16#B,16#C:
	END_CASE
	*)
	
	IF (SIf.stErr.bolErrorActive = FALSE) THEN
		SIf.stErr.bolErrorActive:= TRUE;	
		SIf.stErr.bolSensorError:= TRUE; 
		SIf.stErr.udiErrorID := bytErrorID;	
		// Try to close the socket. Needs reconnect for socket after an error!	
		stStateMachine.intStateNext := cBCD_STA_CloseSocketBusy;	
	END_IF	

END_IF
	
                      
END_METHOD

{attribute 'object_name' := 'sta_ReadCodeBusy'}
METHOD sta_ReadCodeBusy : BOOL
                        // state implemetation
//--------------------------------------------------------------------------------------
// Entry action
	IF (stStateMachine.intState<>stStateMachine.intStateLastCycle) THEN
		stStateMachine.intStateHistory := stStateMachine.intStateLastCycle;
		stStateMachine.intStateLastCycle := stStateMachine.intState;
		
		// Clear data
		SIf.stData.uliBarCode:=0;
		SIf.stData.strBarCode:='';
		SIf.stData.bolCodeReaded:= FALSE;
						
		// Init sub state machine
		stSubStateMachine.intState := cBCD_SUB_Send;
		stSubStateMachine.intStateNext := cBCD_SUB_Send;	
	END_IF

//--------------------------------------------------------------------------------------
// Cyclic action
	IF (stStateMachine.intState=stStateMachine.intStateLastCycle) THEN
			
		// sub state machine for reading the bar code	
		CASE stSubStateMachine.intState OF

			cBCD_SUB_Send:
				// Check Tx state idle
				IF (intTxState = cTxIdle) THEN
					CASE SIf.stCfg.iSensorType OF
						E_BCD_Type.SICK:
							THIS^.PrepareSendMsg('sMN mTCgateon'); // Call SOPAS method "sMN mTCgateon"
							bolExecuteSend:= TRUE;
							stSubStateMachine.intState := cBCD_SUB_Wait;
							
						E_BCD_Type.KEYENCE:
							THIS^.PrepareSendMsg('LON'); // Call Trigger ON
							bolExecuteSend:= TRUE;
							stSubStateMachine.intState := cBCD_SUB_Wait;
					ELSE
						SIf.stData.strBarCode:= 'no sensor type defined';
						SIf.stData.uliBarCode:= 0;
					END_CASE
					
				END_IF
		
			cBCD_SUB_Wait:
				// Wait until executed -> flag set back to false by method handle TxData
				IF (bolExecuteSend=FALSE)THEN
					stSubStateMachine.intState := cBCD_SUB_Read;
				END_IF
				
			cBCD_SUB_Read:
				// Check Rx state idle
				IF (intRxState = cRxIdle) THEN
					bolExecuteRead:= TRUE;
					stSubStateMachine.intState := cBCD_SUB_CheckAnswer;
				END_IF
			
			cBCD_SUB_CheckAnswer:
				// Wait until executed -> flag set back to false by method handle RxData
				IF (bolExecuteRead=FALSE)THEN				
					// Check about corresponding answer for the called method
					CASE SIf.stCfg.iSensorType OF
						E_BCD_Type.SICK:
							IF (FC_StrComp(strReceivedMessage,'sAN mTCgateon 1') = 0) THEN			
								// Check Rx state idle
								IF (intRxState = cRxIdle) THEN
									bolExecuteRead:= TRUE;
									stSubStateMachine.intState := cBCD_SUB_GetData;
								END_IF
							END_IF
							
						E_BCD_Type.KEYENCE:
							IF (FC_StrComp(strReceivedMessage,'OK,LON') = 0) THEN			
								// Check Rx state idle
								IF (intRxState = cRxIdle) THEN
									bolExecuteRead:= TRUE;
									stSubStateMachine.intState := cBCD_SUB_GetData;
								END_IF
							END_IF
					END_CASE
				END_IF
			
			cBCD_SUB_GetData:
				// Wait until executed -> flag set back to false by method handle RxData
				IF (bolExecuteRead=FALSE)THEN
					
					CASE SIf.stCfg.iSensorType OF
						E_BCD_Type.SICK:
							// No barcode recognized after the end of the time window ("duration" setting of sensor object trigger), NoRead !
							IF (((TC2_STANDARD.FIND(strReceivedMessage,'OI=') <> 0) OR NOT SIf.stCfg.bolResponseIncludingDiagnostics) 
								AND (TC2_STANDARD.FIND(strReceivedMessage,'*NoRead*') <> 0)) THEN			
								SIf.stData.strBarCode:='NoRead';
								stSubStateMachine.intState := cBCD_SUB_Done;
							END_IF
							
							// Barcode detected within the time window
							IF (((TC2_STANDARD.FIND(strReceivedMessage,'OI=') <> 0) OR NOT SIf.stCfg.bolResponseIncludingDiagnostics) 
								AND NOT (TC2_STANDARD.FIND(strReceivedMessage,'*NoRead*') <> 0)) THEN			
								// Prepare bar code data from received message
								THIS^.PrepareBarCodeData();
								stSubStateMachine.intState := cBCD_SUB_Done;
							END_IF
						
						E_BCD_Type.KEYENCE:
							// No barcode recognized after the end of the time window ("duration" setting of sensor object trigger), NoRead !
							IF (TC2_STANDARD.FIND(strReceivedMessage,'ERROR') <> 0) THEN			
								SIf.stData.strBarCode:='NoRead';
								stSubStateMachine.intState := cBCD_SUB_Done;
							END_IF
							
							// Barcode detected within the time window
							IF NOT (TC2_STANDARD.FIND(strReceivedMessage,'ERROR') <> 0) THEN			
								// Prepare bar code data from received message
								iStringLength := Tc2_Standard.LEN(strReceivedMessage);
								SIf.stData.strBarCode := Tc2_Standard.LEFT(strReceivedMessage,iStringLength-1);
								SIf.stData.uliBarCode:= STRING_TO_ULINT(SIf.stData.strBarCode);
								stSubStateMachine.intState := cBCD_SUB_Done;
							END_IF
					END_CASE
				END_IF
			
			cBCD_SUB_Done:
				; // job executed
			
		END_CASE
		
		 // job executed
		IF (stSubStateMachine.intState = cBCD_SUB_Done) THEN
			stStateMachine.intStateNext := cBCD_STA_WaitForJob;	
		END_IF
			
	END_IF

//--------------------------------------------------------------------------------------
// Exit action
	IF (stStateMachine.intState<>stStateMachine.intStateNext) THEN
		SIf.intCmd := cBCD_CMD_DONE;
	END_IF
                      
END_METHOD

{attribute 'object_name' := 'PrepareSendMsg'}
METHOD PrepareSendMsg
  VAR_INPUT
    strMsg : STRING;
  END_VAR
  VAR
    intI : UINT;
    strCharacter : STRING(1);
  END_VAR
                        // Clear send buffer
ClearTxBuffer();

// STX - start of telegramm
rTxData.aTxData[0]:= cSTX;

// Loop over message string and convert to ASCII
FOR intI:= 1 TO INT_TO_UINT(LEN(strMsg)) DO
	// Get char
	strCharacter:= MID(strMsg,1,UINT_TO_INT(intI));
	// Convert to ASCII
	rTxData.aTxData[intI]:= F_ToASC(strCharacter);
END_FOR

// ETX - end of telegramm
rTxData.aTxData[intI]:= cETX;

rTxData.intMessageSize := intI + 1;
                      
END_METHOD

{attribute 'object_name' := 'sta_WaitForJob'}
METHOD sta_WaitForJob : BOOL
                        // state implemetation
//--------------------------------------------------------------------------------------
// Entry action
	IF (stStateMachine.intState<>stStateMachine.intStateLastCycle) THEN
		stStateMachine.intStateLastCycle := stStateMachine.intState;
	END_IF


//--------------------------------------------------------------------------------------
// Cyclic action
	IF (stStateMachine.intState=stStateMachine.intStateLastCycle) THEN

		// State Change Condition
		IF (SIf.intCmd=cBCD_CMD_CONNECT_SOCKET) THEN						// Connect TCP socket
			stStateMachine.intStateNext := cBCD_STA_ConnectSocketBusy;
		ELSIF (SIf.intCmd=cBCD_CMD_CLOSE_SOCKET) THEN						// Close TCP socket
			stStateMachine.intStateNext := cBCD_STA_CloseSocketBusy;
		ELSIF (SIf.intCmd=cBCD_CMD_COM_TEST) THEN							// Communication test 
			stStateMachine.intStateNext := cBCD_STA_ComTestBusy;	
		ELSIF (SIf.intCmd=cBCD_CMD_READ_BARCODE) THEN						// Read bar code
			stStateMachine.intStateNext := cBCD_STA_ReadCodeBusy;				
		END_IF

				
	END_IF

//--------------------------------------------------------------------------------------
// Exit action
	IF (stStateMachine.intState<>stStateMachine.intStateNext) THEN
		;
	END_IF
                      
END_METHOD

{attribute 'object_name' := 'CtrlInit'}
METHOD CtrlInit : BOOL
                        // one time first cyclic call
// The socket is closed
stStateMachine.intStateNext := cBCD_STA_SocketClosed;
                      
END_METHOD
END_FUNCTION_BLOCK

FUNCTION FC_StrComp : DINT
  VAR_INPUT
    strArg1 : STRING(255);
    strArg2 : STRING(255);
  END_VAR
  VAR
    stArg1 : TC2_UTILITIES.T_Arg;
    stArg2 : TC2_UTILITIES.T_Arg;
  END_VAR

                  
// String compare function use F_ARGCMP from beckhoff lib. TC2_UTILITIES

// set parameter for arg1
stArg1.cbLen:= INT_TO_UDINT(TC2_STANDARD.LEN(strArg1));
stArg1.pData:= ADR(strArg1);
stArg1.eType:= ARGTYPE_STRING;

// set parameter for arg2
stArg2.cbLen:= INT_TO_UDINT(TC2_STANDARD.LEN(strArg2));
stArg2.pData:= ADR(strArg2);
stArg2.eType:= ARGTYPE_STRING;

// call F_ARGCMP
FC_StrComp:= TC2_UTILITIES.F_ARGCMP(TRUE,stArg1,stArg2);
                
END_FUNCTION

FUNCTION_BLOCK FB_PRS EXTENDS FB_CtrlBase
  VAR_INPUT
    In_bolPresent : BOOL;
  END_VAR
  VAR_OUTPUT
    Out_bolPresent : BOOL;
  END_VAR
  VAR
    SIf : T_Ctrl_SIf_PRS;  (* Specific interface struct for public access *)
  END_VAR

                  (*__________________________________________________________________________________________________
¦	
¦	Vistaprint Schweiz GmbH
¦	CH - 8401 Winterthur
¦
¦	www.vistaprint.ch - info@vistaprint.ch
¦___________________________________________________________________________________________________

Function desription:
Vacuum Pump implementation. 


History:
Version		Date			Author		Comment
---------------------------------------------------------------------------------------------------
0.00.1		09.07.2013		PC			Start history
___________________________________________________________________________________________________*)


IF (me.bolActivate) THEN // cyclic call enabled
	IF (CIf.Info.bolInitDone=FALSE) THEN // first cycle -> init
		CtrlInit();
		CIf.Info.bolInitDone := TRUE;
	ELSE
		CycleStartDuty();
	
		Always();
		
